LIN {X 0,Y 530.709,Z 614.143,A -85,B 0,C 180,E1 -4418.184,E2 -4418.184} C_VEL
LIN {X 0,Y 530.928,Z 606.171,A -85,B 0,C 180,E1 -4419.524,E2 -4419.524} C_VEL
LIN {X 0,Y 531.122,Z 597.851,A -85,B 0,C 180,E1 -4420.676,E2 -4420.676} C_VEL
LIN {X 0,Y 531.454,Z 587.351,A -85,B 0,C 180,E1 -4421.879,E2 -4421.879} C_VEL
LIN {X 0,Y 531.719,Z 576.624,A -85,B 0,C 180,E1 -4422.888,E2 -4422.888} C_VEL
LIN {X 0,Y 532.051,Z 564.106,A -85,B 0,C 180,E1 -4423.852,E2 -4423.852} C_VEL
LIN {X 0,Y 532.469,Z 551.67,A -85,B 0,C 180,E1 -4424.621,E2 -4424.621} C_VEL
LIN {X 0,Y 532.792,Z 537.759,A -85,B 0,C 180,E1 -4425.297,E2 -4425.297} C_VEL
LIN {X 0,Y 533.028,Z 523.286,A -85,B 0,C 180,E1 -4425.814,E2 -4425.814} C_VEL
LIN {X 0,Y 533.143,Z 514.195,A -85,B 0,C 180,E1 -4426.054,E2 -4426.054} C_VEL
LIN {X 0,Y 530.757,Z 502.42,A -85,B 0,C 180,E1 -4426.367,E2 -4426.367} C_VEL
LIN {X 0,Y 530.873,Z 494.542,A -85,B 0,C 180,E1 -4428.926,E2 -4428.926} C_VEL
LIN {X 0,Y 531.011,Z 485.976,A -85,B 0,C 180,E1 -4431.752,E2 -4431.752} C_VEL
LIN {X 0,Y 531.173,Z 477.41,A -85,B 0,C 180,E1 -4434.631,E2 -4434.631} C_VEL
LIN {X 0,Y 531.332,Z 470.067,A -85,B 0,C 180,E1 -4437.151,E2 -4437.151} C_VEL
LIN {X 0,Y 531.503,Z 463.949,A -85,B 0,C 180,E1 -4439.291,E2 -4439.291} C_VEL
LIN {X 0,Y 531.665,Z 455.312,A -85,B 0,C 180,E1 -4442.22,E2 -4442.22} C_VEL
LIN {X 0,Y 531.758,Z 447.204,A -85,B 0,C 180,E1 -4444.973,E2 -4444.973} C_VEL
LIN {X 0,Y 531.783,Z 438.711,A -85,B 0,C 180,E1 -4447.929,E2 -4447.929} C_VEL
LIN {X 0,Y 531.886,Z 429.937,A -85,B 0,C 180,E1 -4451.135,E2 -4451.135} C_VEL
LIN {X 0,Y 532.132,Z 421.148,A -85,B 0,C 180,E1 -4454.505,E2 -4454.505} C_VEL
LIN {X 0,Y 532.173,Z 415.877,A -85,B 0,C 180,E1 -4456.629,E2 -4456.629} C_VEL
LIN {X 0,Y 531.598,Z 411.207,A -85,B 0,C 180,E1 -4458.622,E2 -4458.622} C_VEL
LIN {X 0,Y 530.99,Z 407.971,A -85,B 0,C 180,E1 -4460.145,E2 -4460.145} C_VEL
LIN {X 0,Y 530.968,Z 407.972,A -85,B 0,C 180,E1 -4463.442,E2 -4463.442} C_VEL
LIN {X 0,Y 531.001,Z 407.967,A -85,B 0,C 180,E1 -4466.494,E2 -4466.494} C_VEL
LIN {X 0,Y 530.976,Z 407.969,A -85,B 0,C 180,E1 -4469.355,E2 -4469.355} C_VEL
LIN {X 0,Y 531.017,Z 407.964,A -85,B 0,C 180,E1 -4472.467,E2 -4472.467} C_VEL
LIN {X 0,Y 531.008,Z 407.963,A -85,B 0,C 180,E1 -4474.943,E2 -4474.943} C_VEL
LIN {X 0,Y 530.974,Z 407.967,A -85,B 0,C 180,E1 -4478.247,E2 -4478.247} C_VEL
LIN {X 0,Y 530.999,Z 407.967,A -85,B 0,C 180,E1 -4480.677,E2 -4480.677} C_VEL
LIN {X 0,Y 530.99,Z 407.968,A -85,B 0,C 180,E1 -4483.071,E2 -4483.071} C_VEL
LIN {X 0,Y 531.022,Z 407.959,A -85,B 0,C 180,E1 -4485.436,E2 -4485.436} C_VEL
LIN {X 0,Y 531.039,Z 407.96,A -85,B 0,C 180,E1 -4488.55,E2 -4488.55} C_VEL
LIN {X 0,Y 531.041,Z 407.957,A -85,B 0,C 180,E1 -4491.629,E2 -4491.629} C_VEL
LIN {X 0,Y 531.125,Z 407.95,A -85,B 0,C 180,E1 -4494.685,E2 -4494.685} C_VEL
LIN {X 0,Y 531.14,Z 407.944,A -85,B 0,C 180,E1 -4497.725,E2 -4497.725} C_VEL
LIN {X 0,Y 531.155,Z 407.946,A -85,B 0,C 180,E1 -4500.758,E2 -4500.758} C_VEL
LIN {X 0,Y 531.108,Z 407.951,A -85,B 0,C 180,E1 -4503.034,E2 -4503.034} C_VEL
LIN {X 0,Y 531.086,Z 407.959,A -85,B 0,C 180,E1 -4506.077,E2 -4506.077} C_VEL
LIN {X 0,Y 531.033,Z 407.962,A -85,B 0,C 180,E1 -4509.138,E2 -4509.138} C_VEL
LIN {X 0,Y 531.043,Z 407.962,A -85,B 0,C 180,E1 -4512.225,E2 -4512.225} C_VEL
LIN {X 0,Y 530.999,Z 407.968,A -85,B 0,C 180,E1 -4515.35,E2 -4515.35} C_VEL
LIN {X 0,Y 530.992,Z 407.964,A -85,B 0,C 180,E1 -4518.521,E2 -4518.521} C_VEL
LIN {X 0,Y 531.003,Z 407.969,A -85,B 0,C 180,E1 -4520.938,E2 -4520.938} C_VEL
LIN {X 0,Y 530.968,Z 407.973,A -85,B 0,C 180,E1 -4524.225,E2 -4524.225} C_VEL
LIN {X 0,Y 531.008,Z 407.964,A -85,B 0,C 180,E1 -4526.744,E2 -4526.744} C_VEL
LIN {X 0,Y 530.984,Z 407.967,A -85,B 0,C 180,E1 -4529.323,E2 -4529.323} C_VEL
LIN {X 0,Y 530.968,Z 407.97,A -85,B 0,C 180,E1 -4532.1,E2 -4532.1} C_VEL
LIN {X 0,Y 530.972,Z 407.971,A -85,B 0,C 180,E1 -4534.851,E2 -4534.851} C_VEL
LIN {X 0,Y 530.968,Z 407.974,A -85,B 0,C 180,E1 -4537.508,E2 -4537.508} C_VEL
LIN {X 0,Y 530.984,Z 407.971,A -85,B 0,C 180,E1 -4540.433,E2 -4540.433} C_VEL
LIN {X 0,Y 530.969,Z 407.973,A -85,B 0,C 180,E1 -4543.494,E2 -4543.494} C_VEL
LIN {X 0,Y 530.966,Z 407.973,A -85,B 0,C 180,E1 -4543.565,E2 -4543.565} C_VEL
LIN {X 0,Y 530.293,Z 408.054,A -85,B 0,C 180,E1 -4544.198,E2 -4544.198} C_VEL
LIN {X 0,Y 527.445,Z 408.413,A -85,B 0,C 180,E1 -4545.227,E2 -4545.227} C_VEL
LIN {X 0,Y 525.041,Z 408.716,A -85,B 0,C 180,E1 -4546.056,E2 -4546.056} C_VEL
LIN {X 0,Y 524.007,Z 408.843,A -85,B 0,C 180,E1 -4546.695,E2 -4546.695} C_VEL
LIN {X 0,Y 523.922,Z 408.852,A -85,B 0,C 180,E1 -4546.912,E2 -4546.912} C_VEL
LIN {X 0,Y 523.951,Z 408.848,A -85,B 0,C 180,E1 -4549.921,E2 -4549.921} C_VEL
LIN {X 0,Y 523.963,Z 408.854,A -85,B 0,C 180,E1 -4550.422,E2 -4550.422} C_VEL
LIN {X 0,Y 524.799,Z 414.518,A -85,B 0,C 180,E1 -4551.974,E2 -4551.974} C_VEL
LIN {X 0,Y 524.708,Z 423.272,A -85,B 0,C 180,E1 -4554.364,E2 -4554.364} C_VEL
LIN {X 0,Y 524.58,Z 434.74,A -85,B 0,C 180,E1 -4557.595,E2 -4557.595} C_VEL
LIN {X 0,Y 524.507,Z 445.196,A -85,B 0,C 180,E1 -4560.57,E2 -4560.57} C_VEL
LIN {X 0,Y 524.401,Z 454.996,A -85,B 0,C 180,E1 -4563.323,E2 -4563.323} C_VEL
LIN {X 0,Y 524.205,Z 465.688,A -85,B 0,C 180,E1 -4566.284,E2 -4566.284} C_VEL
LIN {X 0,Y 524.084,Z 476.206,A -85,B 0,C 180,E1 -4569.184,E2 -4569.184} C_VEL
LIN {X 0,Y 523.92,Z 487.271,A -85,B 0,C 180,E1 -4572.254,E2 -4572.254} C_VEL
LIN {X 0,Y 523.813,Z 491.641,A -85,B 0,C 180,E1 -4573.46,E2 -4573.46} C_VEL
LIN {X 0,Y 526.379,Z 504.566,A -85,B 0,C 180,E1 -4573.792,E2 -4573.792} C_VEL
LIN {X 0,Y 526.096,Z 519.046,A -85,B 0,C 180,E1 -4574.209,E2 -4574.209} C_VEL
LIN {X 0,Y 525.838,Z 532.206,A -85,B 0,C 180,E1 -4574.744,E2 -4574.744} C_VEL
LIN {X 0,Y 525.47,Z 545.972,A -85,B 0,C 180,E1 -4575.477,E2 -4575.477} C_VEL
LIN {X 0,Y 525.091,Z 557.559,A -85,B 0,C 180,E1 -4576.257,E2 -4576.257} C_VEL
LIN {X 0,Y 524.696,Z 569.44,A -85,B 0,C 180,E1 -4577.232,E2 -4577.232} C_VEL
LIN {X 0,Y 524.301,Z 580.988,A -85,B 0,C 180,E1 -4578.401,E2 -4578.401} C_VEL
LIN {X 0,Y 524.013,Z 590.481,A -85,B 0,C 180,E1 -4579.568,E2 -4579.568} C_VEL
LIN {X 0,Y 523.762,Z 599.542,A -85,B 0,C 180,E1 -4580.929,E2 -4580.929} C_VEL
LIN {X 0,Y 523.573,Z 606.843,A -85,B 0,C 180,E1 -4582.286,E2 -4582.286} C_VEL
LIN {X 0,Y 523.469,Z 613.433,A -85,B 0,C 180,E1 -4583.834,E2 -4583.834} C_VEL
LIN {X 0,Y 523.353,Z 618.327,A -85,B 0,C 180,E1 -4585.379,E2 -4585.379} C_VEL
LIN {X 0,Y 523.419,Z 620.227,A -85,B 0,C 180,E1 -4586.151,E2 -4586.151} C_VEL
LIN {X 0,Y 523.334,Z 622.94,A -85,B 0,C 180,E1 -4587.691,E2 -4587.691} C_VEL
LIN {X 0,Y 523.246,Z 624.299,A -85,B 0,C 180,E1 -4589.23,E2 -4589.23} C_VEL
LIN {X 0,Y 523.247,Z 624.346,A -85,B 0,C 180,E1 -4590.77,E2 -4590.77} C_VEL
LIN {X 0,Y 523.333,Z 623.049,A -85,B 0,C 180,E1 -4592.309,E2 -4592.309} C_VEL
LIN {X 0,Y 523.42,Z 620.43,A -85,B 0,C 180,E1 -4593.849,E2 -4593.849} C_VEL
LIN {X 0,Y 523.45,Z 616.35,A -85,B 0,C 180,E1 -4595.393,E2 -4595.393} C_VEL
LIN {X 0,Y 523.493,Z 612.29,A -85,B 0,C 180,E1 -4596.552,E2 -4596.552} C_VEL
LIN {X 0,Y 523.568,Z 607.269,A -85,B 0,C 180,E1 -4597.714,E2 -4597.714} C_VEL
LIN {X 0,Y 523.751,Z 600.085,A -85,B 0,C 180,E1 -4599.072,E2 -4599.072} C_VEL
LIN {X 0,Y 524.001,Z 591.128,A -85,B 0,C 180,E1 -4600.432,E2 -4600.432} C_VEL
LIN {X 0,Y 524.308,Z 581.8,A -85,B 0,C 180,E1 -4601.599,E2 -4601.599} C_VEL
LIN {X 0,Y 524.674,Z 570.39,A -85,B 0,C 180,E1 -4602.769,E2 -4602.769} C_VEL
LIN {X 0,Y 525.039,Z 558.753,A -85,B 0,C 180,E1 -4603.745,E2 -4603.745} C_VEL
LIN {X 0,Y 525.479,Z 545.827,A -85,B 0,C 180,E1 -4604.622,E2 -4604.622} C_VEL
LIN {X 0,Y 525.81,Z 532.013,A -85,B 0,C 180,E1 -4605.356,E2 -4605.356} C_VEL
LIN {X 0,Y 526.176,Z 517.48,A -85,B 0,C 180,E1 -4605.933,E2 -4605.933} C_VEL
LIN {X 0,Y 526.361,Z 504.166,A -85,B 0,C 180,E1 -4606.309,E2 -4606.309} C_VEL
LIN {X 0,Y 523.813,Z 491.588,A -85,B 0,C 180,E1 -4606.641,E2 -4606.641} C_VEL
LIN {X 0,Y 523.994,Z 480.988,A -85,B 0,C 180,E1 -4609.591,E2 -4609.591} C_VEL
LIN {X 0,Y 524.186,Z 470.27,A -85,B 0,C 180,E1 -4612.546,E2 -4612.546} C_VEL
LIN {X 0,Y 524.326,Z 458.655,A -85,B 0,C 180,E1 -4615.751,E2 -4615.751} C_VEL
LIN {X 0,Y 524.456,Z 449.135,A -85,B 0,C 180,E1 -4618.406,E2 -4618.406} C_VEL
LIN {X 0,Y 524.576,Z 438.248,A -85,B 0,C 180,E1 -4621.5,E2 -4621.5} C_VEL
LIN {X 0,Y 524.624,Z 428.598,A -85,B 0,C 180,E1 -4624.239,E2 -4624.239} C_VEL
LIN {X 0,Y 524.803,Z 418.429,A -85,B 0,C 180,E1 -4627.058,E2 -4627.058} C_VEL
LIN {X 0,Y 524.689,Z 413.124,A -85,B 0,C 180,E1 -4628.497,E2 -4628.497} C_VEL
LIN {X 0,Y 523.947,Z 408.849,A -85,B 0,C 180,E1 -4629.704,E2 -4629.704} C_VEL
LIN {X 0,Y 523.94,Z 408.849,A -85,B 0,C 180,E1 -4632.459,E2 -4632.459} C_VEL
LIN {X 0,Y 523.959,Z 408.846,A -85,B 0,C 180,E1 -4635.309,E2 -4635.309} C_VEL
LIN {X 0,Y 523.961,Z 408.847,A -85,B 0,C 180,E1 -4638.689,E2 -4638.689} C_VEL
LIN {X 0,Y 523.919,Z 408.851,A -85,B 0,C 180,E1 -4641.081,E2 -4641.081} C_VEL
LIN {X 0,Y 523.929,Z 408.848,A -85,B 0,C 180,E1 -4643.827,E2 -4643.827} C_VEL
LIN {X 0,Y 523.944,Z 408.846,A -85,B 0,C 180,E1 -4646.636,E2 -4646.636} C_VEL
LIN {X 0,Y 523.966,Z 408.84,A -85,B 0,C 180,E1 -4649.356,E2 -4649.356} C_VEL
LIN {X 0,Y 523.979,Z 408.842,A -85,B 0,C 180,E1 -4652.281,E2 -4652.281} C_VEL
LIN {X 0,Y 523.955,Z 408.844,A -85,B 0,C 180,E1 -4654.581,E2 -4654.581} C_VEL
LIN {X 0,Y 523.92,Z 408.849,A -85,B 0,C 180,E1 -4657.107,E2 -4657.107} C_VEL
LIN {X 0,Y 523.982,Z 408.845,A -85,B 0,C 180,E1 -4659.866,E2 -4659.866} C_VEL
LIN {X 0,Y 523.963,Z 408.851,A -85,B 0,C 180,E1 -4661.417,E2 -4661.417} C_VEL
LIN {X 0,Y 526.697,Z 417.552,A -85,B 0,C 180,E1 -4661.826,E2 -4661.826} C_VEL
LIN {X 0,Y 526.634,Z 428.886,A -85,B 0,C 180,E1 -4662.326,E2 -4662.326} C_VEL
LIN {X 0,Y 526.283,Z 440.14,A -85,B 0,C 180,E1 -4662.915,E2 -4662.915} C_VEL
LIN {X 0,Y 525.888,Z 451.09,A -85,B 0,C 180,E1 -4663.601,E2 -4663.601} C_VEL
LIN {X 0,Y 525.483,Z 461.333,A -85,B 0,C 180,E1 -4664.356,E2 -4664.356} C_VEL
LIN {X 0,Y 525.097,Z 470.829,A -85,B 0,C 180,E1 -4665.17,E2 -4665.17} C_VEL
LIN {X 0,Y 524.748,Z 479.724,A -85,B 0,C 180,E1 -4666.05,E2 -4666.05} C_VEL
LIN {X 0,Y 524.46,Z 488.326,A -85,B 0,C 180,E1 -4667.029,E2 -4667.029} C_VEL
LIN {X 0,Y 524.085,Z 497.442,A -85,B 0,C 180,E1 -4668.219,E2 -4668.219} C_VEL
LIN {X 0,Y 523.917,Z 506.187,A -85,B 0,C 180,E1 -4669.566,E2 -4669.566} C_VEL
LIN {X 0,Y 523.66,Z 514.361,A -85,B 0,C 180,E1 -4671.121,E2 -4671.121} C_VEL
LIN {X 0,Y 523.546,Z 519.47,A -85,B 0,C 180,E1 -4672.285,E2 -4672.285} C_VEL
LIN {X 0,Y 523.467,Z 523.823,A -85,B 0,C 180,E1 -4673.472,E2 -4673.472} C_VEL
LIN {X 0,Y 523.441,Z 527.259,A -85,B 0,C 180,E1 -4674.607,E2 -4674.607} C_VEL
LIN {X 0,Y 523.402,Z 530.761,A -85,B 0,C 180,E1 -4676.15,E2 -4676.15} C_VEL
LIN {X 0,Y 523.359,Z 532.149,A -85,B 0,C 180,E1 -4676.921,E2 -4676.921} C_VEL
LIN {X 0,Y 523.27,Z 533.858,A -85,B 0,C 180,E1 -4678.461,E2 -4678.461} C_VEL
LIN {X 0,Y 523.244,Z 534.43,A -85,B 0,C 180,E1 -4680,E2 -4680} C_VEL
LIN {X 0,Y 523.248,Z 534.369,A -85,B 0,C 180,E1 -4680.77,E2 -4680.77} C_VEL
LIN {X 0,Y 523.332,Z 533.247,A -85,B 0,C 180,E1 -4682.309,E2 -4682.309} C_VEL
LIN {X 0,Y 523.403,Z 530.941,A -85,B 0,C 180,E1 -4683.85,E2 -4683.85} C_VEL
LIN {X 0,Y 523.322,Z 529.424,A -85,B 0,C 180,E1 -4684.622,E2 -4684.622} C_VEL
LIN {X 0,Y 523.447,Z 525.299,A -85,B 0,C 180,E1 -4686.166,E2 -4686.166} C_VEL
LIN {X 0,Y 523.533,Z 519.815,A -85,B 0,C 180,E1 -4687.715,E2 -4687.715} C_VEL
LIN {X 0,Y 523.643,Z 514.778,A -85,B 0,C 180,E1 -4688.879,E2 -4688.879} C_VEL
LIN {X 0,Y 523.773,Z 508.825,A -85,B 0,C 180,E1 -4690.046,E2 -4690.046} C_VEL
LIN {X 0,Y 524.03,Z 501.839,A -85,B 0,C 180,E1 -4691.213,E2 -4691.213} C_VEL
LIN {X 0,Y 524.203,Z 495.095,A -85,B 0,C 180,E1 -4692.194,E2 -4692.194} C_VEL
LIN {X 0,Y 524.48,Z 487.449,A -85,B 0,C 180,E1 -4693.167,E2 -4693.167} C_VEL
LIN {X 0,Y 524.814,Z 478.744,A -85,B 0,C 180,E1 -4694.146,E2 -4694.146} C_VEL
LIN {X 0,Y 525.139,Z 469.8,A -85,B 0,C 180,E1 -4695.019,E2 -4695.019} C_VEL
LIN {X 0,Y 525.609,Z 459.629,A -85,B 0,C 180,E1 -4695.869,E2 -4695.869} C_VEL
LIN {X 0,Y 525.986,Z 448.044,A -85,B 0,C 180,E1 -4696.695,E2 -4696.695} C_VEL
LIN {X 0,Y 526.476,Z 434.632,A -85,B 0,C 180,E1 -4697.479,E2 -4697.479} C_VEL
LIN {X 0,Y 526.827,Z 420.353,A -85,B 0,C 180,E1 -4698.132,E2 -4698.132} C_VEL
LIN {X 0,Y 526.605,Z 417.439,A -85,B 0,C 180,E1 -4698.258,E2 -4698.258} C_VEL
LIN {X 0,Y 523.963,Z 408.843,A -85,B 0,C 180,E1 -4698.655,E2 -4698.655} C_VEL
LIN {X 0,Y 523.948,Z 408.843,A -85,B 0,C 180,E1 -4701.233,E2 -4701.233} C_VEL
LIN {X 0,Y 523.928,Z 408.847,A -85,B 0,C 180,E1 -4704.572,E2 -4704.572} C_VEL
LIN {X 0,Y 523.956,Z 408.842,A -85,B 0,C 180,E1 -4707.133,E2 -4707.133} C_VEL
LIN {X 0,Y 523.945,Z 408.849,A -85,B 0,C 180,E1 -4709.756,E2 -4709.756} C_VEL
LIN {X 0,Y 523.942,Z 408.843,A -85,B 0,C 180,E1 -4712.449,E2 -4712.449} C_VEL
LIN {X 0,Y 523.922,Z 408.847,A -85,B 0,C 180,E1 -4715.227,E2 -4715.227} C_VEL
LIN {X 0,Y 523.917,Z 408.849,A -85,B 0,C 180,E1 -4718.102,E2 -4718.102} C_VEL
LIN {X 0,Y 523.943,Z 408.845,A -85,B 0,C 180,E1 -4721.092,E2 -4721.092} C_VEL
LIN {X 0,Y 523.952,Z 408.846,A -85,B 0,C 180,E1 -4724.227,E2 -4724.227} C_VEL
LIN {X 0,Y 523.997,Z 408.934,A -85,B 0,C 180,E1 -4724.797,E2 -4724.797} C_VEL
LIN {X 0,Y 523.747,Z 419.256,A -85,B 0,C 180,E1 -4727.861,E2 -4727.861} C_VEL
LIN {X 0,Y 524.048,Z 430.498,A -85,B 0,C 180,E1 -4731.063,E2 -4731.063} C_VEL
LIN {X 0,Y 524.288,Z 440.494,A -85,B 0,C 180,E1 -4733.856,E2 -4733.856} C_VEL
LIN {X 0,Y 524.4,Z 448.893,A -85,B 0,C 180,E1 -4736.194,E2 -4736.194} C_VEL
LIN {X 0,Y 524.489,Z 459.131,A -85,B 0,C 180,E1 -4739.046,E2 -4739.046} C_VEL
LIN {X 0,Y 524.528,Z 466.39,A -85,B 0,C 180,E1 -4741.161,E2 -4741.161} C_VEL
LIN {X 0,Y 524.219,Z 476.186,A -85,B 0,C 180,E1 -4744.595,E2 -4744.595} C_VEL
LIN {X 0,Y 523.984,Z 485.381,A -85,B 0,C 180,E1 -4747.74,E2 -4747.74} C_VEL
LIN {X 0,Y 523.869,Z 493.319,A -85,B 0,C 180,E1 -4750.404,E2 -4750.404} C_VEL
LIN {X 0,Y 523.742,Z 502.599,A -85,B 0,C 180,E1 -4753.432,E2 -4753.432} C_VEL
LIN {X 0,Y 526.393,Z 515.813,A -85,B 0,C 180,E1 -4753.774,E2 -4753.774} C_VEL
LIN {X 0,Y 526.109,Z 529.055,A -85,B 0,C 180,E1 -4754.162,E2 -4754.162} C_VEL
LIN {X 0,Y 525.793,Z 543.152,A -85,B 0,C 180,E1 -4754.743,E2 -4754.743} C_VEL
LIN {X 0,Y 525.438,Z 556.679,A -85,B 0,C 180,E1 -4755.476,E2 -4755.476} C_VEL
LIN {X 0,Y 525.001,Z 569.459,A -85,B 0,C 180,E1 -4756.353,E2 -4756.353} C_VEL
LIN {X 0,Y 524.624,Z 580.966,A -85,B 0,C 180,E1 -4757.328,E2 -4757.328} C_VEL
LIN {X 0,Y 524.335,Z 591.384,A -85,B 0,C 180,E1 -4758.401,E2 -4758.401} C_VEL
LIN {X 0,Y 523.997,Z 600.801,A -85,B 0,C 180,E1 -4759.568,E2 -4759.568} C_VEL
LIN {X 0,Y 523.761,Z 609.812,A -85,B 0,C 180,E1 -4760.929,E2 -4760.929} C_VEL
LIN {X 0,Y 523.569,Z 617.068,A -85,B 0,C 180,E1 -4762.286,E2 -4762.286} C_VEL
LIN {X 0,Y 523.468,Z 623.582,A -85,B 0,C 180,E1 -4763.834,E2 -4763.834} C_VEL
LIN {X 0,Y 523.376,Z 627.394,A -85,B 0,C 180,E1 -4764.993,E2 -4764.993} C_VEL
LIN {X 0,Y 523.419,Z 630.314,A -85,B 0,C 180,E1 -4766.151,E2 -4766.151} C_VEL
LIN {X 0,Y 523.333,Z 632.997,A -85,B 0,C 180,E1 -4767.691,E2 -4767.691} C_VEL
LIN {X 0,Y 523.247,Z 634.332,A -85,B 0,C 180,E1 -4769.23,E2 -4769.23} C_VEL
LIN {X 0,Y 523.247,Z 634.331,A -85,B 0,C 180,E1 -4770.77,E2 -4770.77} C_VEL
LIN {X 0,Y 523.333,Z 632.997,A -85,B 0,C 180,E1 -4772.309,E2 -4772.309} C_VEL
LIN {X 0,Y 523.419,Z 630.318,A -85,B 0,C 180,E1 -4773.849,E2 -4773.849} C_VEL
LIN {X 0,Y 523.449,Z 626.217,A -85,B 0,C 180,E1 -4775.393,E2 -4775.393} C_VEL
LIN {X 0,Y 523.495,Z 620.547,A -85,B 0,C 180,E1 -4776.94,E2 -4776.94} C_VEL
LIN {X 0,Y 523.664,Z 614.145,A -85,B 0,C 180,E1 -4778.295,E2 -4778.295} C_VEL
LIN {X 0,Y 523.863,Z 606.17,A -85,B 0,C 180,E1 -4779.654,E2 -4779.654} C_VEL
LIN {X 0,Y 524.115,Z 597.851,A -85,B 0,C 180,E1 -4780.82,E2 -4780.82} C_VEL
LIN {X 0,Y 524.449,Z 587.082,A -85,B 0,C 180,E1 -4782.068,E2 -4782.068} C_VEL
LIN {X 0,Y 524.805,Z 575.469,A -85,B 0,C 180,E1 -4783.159,E2 -4783.159} C_VEL
LIN {X 0,Y 525.179,Z 562.703,A -85,B 0,C 180,E1 -4784.136,E2 -4784.136} C_VEL
LIN {X 0,Y 525.639,Z 549.923,A -85,B 0,C 180,E1 -4784.915,E2 -4784.915} C_VEL
LIN {X 0,Y 525.937,Z 537.761,A -85,B 0,C 180,E1 -4785.501,E2 -4785.501} C_VEL
LIN {X 0,Y 526.206,Z 523.168,A -85,B 0,C 180,E1 -4786.028,E2 -4786.028} C_VEL
LIN {X 0,Y 526.212,Z 514.561,A -85,B 0,C 180,E1 -4786.263,E2 -4786.263} C_VEL
LIN {X 0,Y 523.732,Z 502.42,A -85,B 0,C 180,E1 -4786.593,E2 -4786.593} C_VEL
LIN {X 0,Y 523.869,Z 493.319,A -85,B 0,C 180,E1 -4789.596,E2 -4789.596} C_VEL
LIN {X 0,Y 523.984,Z 485.381,A -85,B 0,C 180,E1 -4792.26,E2 -4792.26} C_VEL
LIN {X 0,Y 524.219,Z 476.186,A -85,B 0,C 180,E1 -4795.405,E2 -4795.405} C_VEL
LIN {X 0,Y 524.528,Z 466.39,A -85,B 0,C 180,E1 -4798.839,E2 -4798.839} C_VEL
LIN {X 0,Y 524.587,Z 457.054,A -85,B 0,C 180,E1 -4801.951,E2 -4801.951} C_VEL
LIN {X 0,Y 524.695,Z 449.048,A -85,B 0,C 180,E1 -4804.699,E2 -4804.699} C_VEL
LIN {X 0,Y 524.763,Z 441.282,A -85,B 0,C 180,E1 -4807.432,E2 -4807.432} C_VEL
LIN {X 0,Y 524.879,Z 433.589,A -85,B 0,C 180,E1 -4810.251,E2 -4810.251} C_VEL
LIN {X 0,Y 524.991,Z 426.262,A -85,B 0,C 180,E1 -4813.058,E2 -4813.058} C_VEL
LIN {X 0,Y 525.253,Z 419.101,A -85,B 0,C 180,E1 -4815.911,E2 -4815.911} C_VEL
LIN {X 0,Y 525.086,Z 415.535,A -85,B 0,C 180,E1 -4817.404,E2 -4817.404} C_VEL
LIN {X 0,Y 524.13,Z 409.809,A -85,B 0,C 180,E1 -4819.937,E2 -4819.937} C_VEL
LIN {X 0,Y 523.95,Z 408.848,A -85,B 0,C 180,E1 -4820.421,E2 -4820.421} C_VEL
LIN {X 0,Y 523.922,Z 408.85,A -85,B 0,C 180,E1 -4823.596,E2 -4823.596} C_VEL
LIN {X 0,Y 523.943,Z 408.847,A -85,B 0,C 180,E1 -4826.636,E2 -4826.636} C_VEL
LIN {X 0,Y 523.957,Z 408.844,A -85,B 0,C 180,E1 -4829.356,E2 -4829.356} C_VEL
LIN {X 0,Y 523.981,Z 408.84,A -85,B 0,C 180,E1 -4832.281,E2 -4832.281} C_VEL
LIN {X 0,Y 523.956,Z 408.844,A -85,B 0,C 180,E1 -4834.581,E2 -4834.581} C_VEL
LIN {X 0,Y 523.92,Z 408.849,A -85,B 0,C 180,E1 -4837.107,E2 -4837.107} C_VEL
LIN {X 0,Y 523.981,Z 408.835,A -85,B 0,C 180,E1 -4839.866,E2 -4839.866} C_VEL
LIN {X 0,Y 523.97,Z 408.841,A -85,B 0,C 180,E1 -4842.837,E2 -4842.837} C_VEL
LIN {X 0,Y 523.979,Z 408.838,A -85,B 0,C 180,E1 -4845.236,E2 -4845.236} C_VEL
LIN {X 0,Y 524.015,Z 408.836,A -85,B 0,C 180,E1 -4848.394,E2 -4848.394} C_VEL
LIN {X 0,Y 523.993,Z 408.834,A -85,B 0,C 180,E1 -4851.516,E2 -4851.516} C_VEL
LIN {X 0,Y 524.086,Z 408.826,A -85,B 0,C 180,E1 -4854.614,E2 -4854.614} C_VEL
LIN {X 0,Y 524.112,Z 408.819,A -85,B 0,C 180,E1 -4857.695,E2 -4857.695} C_VEL
LIN {X 0,Y 524.126,Z 408.821,A -85,B 0,C 180,E1 -4860.768,E2 -4860.768} C_VEL
LIN {X 0,Y 524.074,Z 408.827,A -85,B 0,C 180,E1 -4863.075,E2 -4863.075} C_VEL
LIN {X 0,Y 524.048,Z 408.834,A -85,B 0,C 180,E1 -4866.159,E2 -4866.159} C_VEL
LIN {X 0,Y 524.001,Z 408.838,A -85,B 0,C 180,E1 -4869.262,E2 -4869.262} C_VEL
LIN {X 0,Y 524.005,Z 408.839,A -85,B 0,C 180,E1 -4871.74,E2 -4871.74} C_VEL
LIN {X 0,Y 523.996,Z 408.841,A -85,B 0,C 180,E1 -4875.052,E2 -4875.052} C_VEL
LIN {X 0,Y 523.966,Z 408.844,A -85,B 0,C 180,E1 -4877.969,E2 -4877.969} C_VEL
LIN {X 0,Y 523.975,Z 408.841,A -85,B 0,C 180,E1 -4880.41,E2 -4880.41} C_VEL
LIN {X 0,Y 523.913,Z 408.848,A -85,B 0,C 180,E1 -4882.894,E2 -4882.894} C_VEL
LIN {X 0,Y 523.987,Z 408.838,A -85,B 0,C 180,E1 -4886.02,E2 -4886.02} C_VEL
LIN {X 0,Y 523.942,Z 408.846,A -85,B 0,C 180,E1 -4888.875,E2 -4888.875} C_VEL
LIN {X 0,Y 523.924,Z 408.852,A -85,B 0,C 180,E1 -4891.544,E2 -4891.544} C_VEL
LIN {X 0,Y 523.935,Z 408.847,A -85,B 0,C 180,E1 -4894.29,E2 -4894.29} C_VEL
LIN {X 0,Y 523.909,Z 408.85,A -85,B 0,C 180,E1 -4897.132,E2 -4897.132} C_VEL
LIN {X 0,Y 523.939,Z 408.846,A -85,B 0,C 180,E1 -4900.13,E2 -4900.13} C_VEL
LIN {X 0,Y 523.942,Z 408.847,A -85,B 0,C 180,E1 -4902.459,E2 -4902.459} C_VEL
LIN {X 0,Y 523.959,Z 408.847,A -85,B 0,C 180,E1 -4905.309,E2 -4905.309} C_VEL
LIN {X 0,Y 523.922,Z 408.852,A -85,B 0,C 180,E1 -4906.912,E2 -4906.912} C_VEL
LIN {X 0,Y 523.241,Z 408.936,A -85,B 0,C 180,E1 -4907.34,E2 -4907.34} C_VEL
LIN {X 0,Y 520.398,Z 409.293,A -85,B 0,C 180,E1 -4908.009,E2 -4908.009} C_VEL
LIN {X 0,Y 517.552,Z 409.647,A -85,B 0,C 180,E1 -4908.684,E2 -4908.684} C_VEL
LIN {X 0,Y 516.884,Z 409.729,A -85,B 0,C 180,E1 -4909.12,E2 -4909.12} C_VEL
LIN {X 0,Y 516.955,Z 409.896,A -85,B 0,C 180,E1 -4910.285,E2 -4910.285} C_VEL
LIN {X 0,Y 517.853,Z 415.763,A -85,B 0,C 180,E1 -4911.919,E2 -4911.919} C_VEL
LIN {X 0,Y 517.725,Z 425.224,A -85,B 0,C 180,E1 -4914.537,E2 -4914.537} C_VEL
LIN {X 0,Y 517.577,Z 437.464,A -85,B 0,C 180,E1 -4918.024,E2 -4918.024} C_VEL
LIN {X 0,Y 517.455,Z 446.879,A -85,B 0,C 180,E1 -4920.729,E2 -4920.729} C_VEL
LIN {X 0,Y 517.373,Z 454.607,A -85,B 0,C 180,E1 -4922.931,E2 -4922.931} C_VEL
LIN {X 0,Y 517.176,Z 465.383,A -85,B 0,C 180,E1 -4925.941,E2 -4925.941} C_VEL
LIN {X 0,Y 517.082,Z 474.488,A -85,B 0,C 180,E1 -4928.471,E2 -4928.471} C_VEL
LIN {X 0,Y 516.923,Z 484.937,A -85,B 0,C 180,E1 -4931.367,E2 -4931.367} C_VEL
LIN {X 0,Y 516.779,Z 491.628,A -85,B 0,C 180,E1 -4933.228,E2 -4933.228} C_VEL
LIN {X 0,Y 519.536,Z 505.622,A -85,B 0,C 180,E1 -4933.598,E2 -4933.598} C_VEL
LIN {X 0,Y 519.262,Z 519.612,A -85,B 0,C 180,E1 -4934.015,E2 -4934.015} C_VEL
LIN {X 0,Y 518.954,Z 533.309,A -85,B 0,C 180,E1 -4934.587,E2 -4934.587} C_VEL
LIN {X 0,Y 518.575,Z 546.012,A -85,B 0,C 180,E1 -4935.279,E2 -4935.279} C_VEL
LIN {X 0,Y 518.169,Z 557.633,A -85,B 0,C 180,E1 -4936.069,E2 -4936.069} C_VEL
LIN {X 0,Y 517.732,Z 569.449,A -85,B 0,C 180,E1 -4937.057,E2 -4937.057} C_VEL
LIN {X 0,Y 517.295,Z 580.345,A -85,B 0,C 180,E1 -4938.167,E2 -4938.167} C_VEL
LIN {X 0,Y 517.013,Z 590.492,A -85,B 0,C 180,E1 -4939.426,E2 -4939.426} C_VEL
LIN {X 0,Y 516.731,Z 599.547,A -85,B 0,C 180,E1 -4940.804,E2 -4940.804} C_VEL
LIN {X 0,Y 516.506,Z 606.846,A -85,B 0,C 180,E1 -4942.18,E2 -4942.18} C_VEL
LIN {X 0,Y 516.385,Z 613.437,A -85,B 0,C 180,E1 -4943.749,E2 -4943.749} C_VEL
LIN {X 0,Y 516.306,Z 617.266,A -85,B 0,C 180,E1 -4944.924,E2 -4944.924} C_VEL
LIN {X 0,Y 516.325,Z 620.228,A -85,B 0,C 180,E1 -4946.098,E2 -4946.098} C_VEL
LIN {X 0,Y 516.26,Z 622.939,A -85,B 0,C 180,E1 -4947.659,E2 -4947.659} C_VEL
LIN {X 0,Y 516.156,Z 624.298,A -85,B 0,C 180,E1 -4949.22,E2 -4949.22} C_VEL
LIN {X 0,Y 516.157,Z 624.345,A -85,B 0,C 180,E1 -4950.78,E2 -4950.78} C_VEL
LIN {X 0,Y 516.259,Z 623.046,A -85,B 0,C 180,E1 -4952.341,E2 -4952.341} C_VEL
LIN {X 0,Y 516.325,Z 620.429,A -85,B 0,C 180,E1 -4953.902,E2 -4953.902} C_VEL
LIN {X 0,Y 516.384,Z 616.347,A -85,B 0,C 180,E1 -4955.467,E2 -4955.467} C_VEL
LIN {X 0,Y 516.398,Z 612.708,A -85,B 0,C 180,E1 -4956.533,E2 -4956.533} C_VEL
LIN {X 0,Y 516.499,Z 607.266,A -85,B 0,C 180,E1 -4957.821,E2 -4957.821} C_VEL
LIN {X 0,Y 516.701,Z 600.083,A -85,B 0,C 180,E1 -4959.196,E2 -4959.196} C_VEL
LIN {X 0,Y 516.996,Z 591.153,A -85,B 0,C 180,E1 -4960.575,E2 -4960.575} C_VEL
LIN {X 0,Y 517.326,Z 580.986,A -85,B 0,C 180,E1 -4961.849,E2 -4961.849} C_VEL
LIN {X 0,Y 517.724,Z 570.392,A -85,B 0,C 180,E1 -4962.943,E2 -4962.943} C_VEL
LIN {X 0,Y 518.094,Z 558.767,A -85,B 0,C 180,E1 -4963.933,E2 -4963.933} C_VEL
LIN {X 0,Y 518.537,Z 547.395,A -85,B 0,C 180,E1 -4964.722,E2 -4964.722} C_VEL
LIN {X 0,Y 518.921,Z 534.135,A -85,B 0,C 180,E1 -4965.464,E2 -4965.464} C_VEL
LIN {X 0,Y 519.249,Z 521.235,A -85,B 0,C 180,E1 -4966.018,E2 -4966.018} C_VEL
LIN {X 0,Y 519.559,Z 506.851,A -85,B 0,C 180,E1 -4966.462,E2 -4966.462} C_VEL
LIN {X 0,Y 518.68,Z 500.619,A -85,B 0,C 180,E1 -4966.635,E2 -4966.635} C_VEL
LIN {X 0,Y 516.806,Z 491.575,A -85,B 0,C 180,E1 -4966.873,E2 -4966.873} C_VEL
LIN {X 0,Y 516.987,Z 480.828,A -85,B 0,C 180,E1 -4969.868,E2 -4969.868} C_VEL
LIN {X 0,Y 517.143,Z 470.286,A -85,B 0,C 180,E1 -4972.787,E2 -4972.787} C_VEL
LIN {X 0,Y 517.281,Z 459.55,A -85,B 0,C 180,E1 -4975.77,E2 -4975.77} C_VEL
LIN {X 0,Y 517.439,Z 450.29,A -85,B 0,C 180,E1 -4978.384,E2 -4978.384} C_VEL
LIN {X 0,Y 517.55,Z 440.547,A -85,B 0,C 180,E1 -4981.185,E2 -4981.185} C_VEL
LIN {X 0,Y 517.632,Z 429.382,A -85,B 0,C 180,E1 -4984.382,E2 -4984.382} C_VEL
LIN {X 0,Y 517.85,Z 419.401,A -85,B 0,C 180,E1 -4987.175,E2 -4987.175} C_VEL
LIN {X 0,Y 517.653,Z 414.051,A -85,B 0,C 180,E1 -4988.648,E2 -4988.648} C_VEL
LIN {X 0,Y 516.895,Z 409.728,A -85,B 0,C 180,E1 -4989.908,E2 -4989.908} C_VEL
LIN {X 0,Y 516.887,Z 409.727,A -85,B 0,C 180,E1 -4992.831,E2 -4992.831} C_VEL
LIN {X 0,Y 516.925,Z 409.723,A -85,B 0,C 180,E1 -4995.01,E2 -4995.01} C_VEL
LIN {X 0,Y 516.918,Z 409.725,A -85,B 0,C 180,E1 -4998.398,E2 -4998.398} C_VEL
LIN {X 0,Y 516.882,Z 409.727,A -85,B 0,C 180,E1 -5001.284,E2 -5001.284} C_VEL
LIN {X 0,Y 516.891,Z 409.727,A -85,B 0,C 180,E1 -5004.221,E2 -5004.221} C_VEL
LIN {X 0,Y 516.897,Z 409.724,A -85,B 0,C 180,E1 -5007.053,E2 -5007.053} C_VEL
LIN {X 0,Y 516.903,Z 409.719,A -85,B 0,C 180,E1 -5009.797,E2 -5009.797} C_VEL
LIN {X 0,Y 516.928,Z 409.722,A -85,B 0,C 180,E1 -5012.467,E2 -5012.467} C_VEL
LIN {X 0,Y 516.913,Z 409.724,A -85,B 0,C 180,E1 -5015.072,E2 -5015.072} C_VEL
LIN {X 0,Y 516.873,Z 409.729,A -85,B 0,C 180,E1 -5017.622,E2 -5017.622} C_VEL
LIN {X 0,Y 516.935,Z 409.722,A -85,B 0,C 180,E1 -5020.13,E2 -5020.13} C_VEL
LIN {X 0,Y 516.944,Z 409.786,A -85,B 0,C 180,E1 -5021.195,E2 -5021.195} C_VEL
LIN {X 0,Y 520.053,Z 419.942,A -85,B 0,C 180,E1 -5021.687,E2 -5021.687} C_VEL
LIN {X 0,Y 519.749,Z 432.987,A -85,B 0,C 180,E1 -5022.287,E2 -5022.287} C_VEL
LIN {X 0,Y 519.248,Z 446.951,A -85,B 0,C 180,E1 -5023.082,E2 -5023.082} C_VEL
LIN {X 0,Y 518.741,Z 460.065,A -85,B 0,C 180,E1 -5024.015,E2 -5024.015} C_VEL
LIN {X 0,Y 518.268,Z 470.326,A -85,B 0,C 180,E1 -5024.886,E2 -5024.886} C_VEL
LIN {X 0,Y 517.865,Z 480.169,A -85,B 0,C 180,E1 -5025.861,E2 -5025.861} C_VEL
LIN {X 0,Y 517.553,Z 488.779,A -85,B 0,C 180,E1 -5026.853,E2 -5026.853} C_VEL
LIN {X 0,Y 517.201,Z 496.275,A -85,B 0,C 180,E1 -5027.841,E2 -5027.841} C_VEL
LIN {X 0,Y 517.026,Z 502.798,A -85,B 0,C 180,E1 -5028.831,E2 -5028.831} C_VEL
LIN {X 0,Y 516.714,Z 509.564,A -85,B 0,C 180,E1 -5030.013,E2 -5030.013} C_VEL
LIN {X 0,Y 516.599,Z 514.424,A -85,B 0,C 180,E1 -5030.999,E2 -5030.999} C_VEL
LIN {X 0,Y 516.473,Z 519.465,A -85,B 0,C 180,E1 -5032.179,E2 -5032.179} C_VEL
LIN {X 0,Y 516.371,Z 524.168,A -85,B 0,C 180,E1 -5033.493,E2 -5033.493} C_VEL
LIN {X 0,Y 516.373,Z 527.254,A -85,B 0,C 180,E1 -5034.533,E2 -5034.533} C_VEL
LIN {X 0,Y 516.308,Z 530.758,A -85,B 0,C 180,E1 -5036.097,E2 -5036.097} C_VEL
LIN {X 0,Y 516.272,Z 532.152,A -85,B 0,C 180,E1 -5036.879,E2 -5036.879} C_VEL
LIN {X 0,Y 516.188,Z 533.854,A -85,B 0,C 180,E1 -5038.44,E2 -5038.44} C_VEL
LIN {X 0,Y 516.152,Z 534.424,A -85,B 0,C 180,E1 -5040,E2 -5040} C_VEL
LIN {X 0,Y 516.158,Z 534.37,A -85,B 0,C 180,E1 -5040.78,E2 -5040.78} C_VEL
LIN {X 0,Y 516.258,Z 533.24,A -85,B 0,C 180,E1 -5042.341,E2 -5042.341} C_VEL
LIN {X 0,Y 516.308,Z 530.934,A -85,B 0,C 180,E1 -5043.903,E2 -5043.903} C_VEL
LIN {X 0,Y 516.238,Z 529.421,A -85,B 0,C 180,E1 -5044.685,E2 -5044.685} C_VEL
LIN {X 0,Y 516.372,Z 525.291,A -85,B 0,C 180,E1 -5046.251,E2 -5046.251} C_VEL
LIN {X 0,Y 516.461,Z 519.807,A -85,B 0,C 180,E1 -5047.821,E2 -5047.821} C_VEL
LIN {X 0,Y 516.579,Z 514.853,A -85,B 0,C 180,E1 -5049.001,E2 -5049.001} C_VEL
LIN {X 0,Y 516.755,Z 509.049,A -85,B 0,C 180,E1 -5050.184,E2 -5050.184} C_VEL
LIN {X 0,Y 517.035,Z 502.21,A -85,B 0,C 180,E1 -5051.367,E2 -5051.367} C_VEL
LIN {X 0,Y 517.304,Z 494.187,A -85,B 0,C 180,E1 -5052.555,E2 -5052.555} C_VEL
LIN {X 0,Y 517.723,Z 484.75,A -85,B 0,C 180,E1 -5053.742,E2 -5053.742} C_VEL
LIN {X 0,Y 518.157,Z 473.391,A -85,B 0,C 180,E1 -5054.934,E2 -5054.934} C_VEL
LIN {X 0,Y 518.669,Z 462.264,A -85,B 0,C 180,E1 -5055.905,E2 -5055.905} C_VEL
LIN {X 0,Y 519.123,Z 449.772,A -85,B 0,C 180,E1 -5056.821,E2 -5056.821} C_VEL
LIN {X 0,Y 519.599,Z 436.495,A -85,B 0,C 180,E1 -5057.616,E2 -5057.616} C_VEL
LIN {X 0,Y 519.977,Z 422.263,A -85,B 0,C 180,E1 -5058.288,E2 -5058.288} C_VEL
LIN {X 0,Y 519.934,Z 419.564,A -85,B 0,C 180,E1 -5058.401,E2 -5058.401} C_VEL
LIN {X 0,Y 516.916,Z 409.72,A -85,B 0,C 180,E1 -5058.867,E2 -5058.867} C_VEL
LIN {X 0,Y 516.888,Z 409.725,A -85,B 0,C 180,E1 -5061.538,E2 -5061.538} C_VEL
LIN {X 0,Y 516.884,Z 409.727,A -85,B 0,C 180,E1 -5064.357,E2 -5064.357} C_VEL
LIN {X 0,Y 516.929,Z 409.718,A -85,B 0,C 180,E1 -5066.658,E2 -5066.658} C_VEL
LIN {X 0,Y 516.913,Z 409.724,A -85,B 0,C 180,E1 -5069.524,E2 -5069.524} C_VEL
LIN {X 0,Y 516.903,Z 409.72,A -85,B 0,C 180,E1 -5072.544,E2 -5072.544} C_VEL
LIN {X 0,Y 516.868,Z 409.727,A -85,B 0,C 180,E1 -5075.33,E2 -5075.33} C_VEL
LIN {X 0,Y 516.882,Z 409.727,A -85,B 0,C 180,E1 -5077.943,E2 -5077.943} C_VEL
LIN {X 0,Y 516.886,Z 409.722,A -85,B 0,C 180,E1 -5080.741,E2 -5080.741} C_VEL
LIN {X 0,Y 516.907,Z 409.722,A -85,B 0,C 180,E1 -5082.829,E2 -5082.829} C_VEL
LIN {X 0,Y 516.966,Z 409.844,A -85,B 0,C 180,E1 -5084.711,E2 -5084.711} C_VEL
LIN {X 0,Y 516.708,Z 418.142,A -85,B 0,C 180,E1 -5087.263,E2 -5087.263} C_VEL
LIN {X 0,Y 516.956,Z 430.227,A -85,B 0,C 180,E1 -5090.797,E2 -5090.797} C_VEL
LIN {X 0,Y 517.22,Z 440.677,A -85,B 0,C 180,E1 -5093.776,E2 -5093.776} C_VEL
LIN {X 0,Y 517.333,Z 450.747,A -85,B 0,C 180,E1 -5096.62,E2 -5096.62} C_VEL
LIN {X 0,Y 517.385,Z 460.518,A -85,B 0,C 180,E1 -5099.377,E2 -5099.377} C_VEL
LIN {X 0,Y 517.395,Z 468.367,A -85,B 0,C 180,E1 -5101.613,E2 -5101.613} C_VEL
LIN {X 0,Y 517.282,Z 473.739,A -85,B 0,C 180,E1 -5103.362,E2 -5103.362} C_VEL
LIN {X 0,Y 517.046,Z 482.305,A -85,B 0,C 180,E1 -5106.36,E2 -5106.36} C_VEL
LIN {X 0,Y 516.911,Z 490.871,A -85,B 0,C 180,E1 -5109.298,E2 -5109.298} C_VEL
LIN {X 0,Y 516.704,Z 500.661,A -85,B 0,C 180,E1 -5112.588,E2 -5112.588} C_VEL
LIN {X 0,Y 516.676,Z 502.599,A -85,B 0,C 180,E1 -5113.199,E2 -5113.199} C_VEL
LIN {X 0,Y 519.564,Z 516.699,A -85,B 0,C 180,E1 -5113.578,E2 -5113.578} C_VEL
LIN {X 0,Y 519.233,Z 530.77,A -85,B 0,C 180,E1 -5114.011,E2 -5114.011} C_VEL
LIN {X 0,Y 518.905,Z 544.18,A -85,B 0,C 180,E1 -5114.586,E2 -5114.586} C_VEL
LIN {X 0,Y 518.536,Z 556.679,A -85,B 0,C 180,E1 -5115.278,E2 -5115.278} C_VEL
LIN {X 0,Y 518.069,Z 569.462,A -85,B 0,C 180,E1 -5116.167,E2 -5116.167} C_VEL
LIN {X 0,Y 517.673,Z 580.964,A -85,B 0,C 180,E1 -5117.155,E2 -5117.155} C_VEL
LIN {X 0,Y 517.335,Z 591.382,A -85,B 0,C 180,E1 -5118.242,E2 -5118.242} C_VEL
LIN {X 0,Y 516.994,Z 600.799,A -85,B 0,C 180,E1 -5119.425,E2 -5119.425} C_VEL
LIN {X 0,Y 516.71,Z 609.811,A -85,B 0,C 180,E1 -5120.804,E2 -5120.804} C_VEL
LIN {X 0,Y 516.501,Z 617.069,A -85,B 0,C 180,E1 -5122.18,E2 -5122.18} C_VEL
LIN {X 0,Y 516.385,Z 623.582,A -85,B 0,C 180,E1 -5123.749,E2 -5123.749} C_VEL
LIN {X 0,Y 516.306,Z 627.395,A -85,B 0,C 180,E1 -5124.924,E2 -5124.924} C_VEL
LIN {X 0,Y 516.324,Z 630.313,A -85,B 0,C 180,E1 -5126.098,E2 -5126.098} C_VEL
LIN {X 0,Y 516.259,Z 632.997,A -85,B 0,C 180,E1 -5127.659,E2 -5127.659} C_VEL
LIN {X 0,Y 516.157,Z 634.332,A -85,B 0,C 180,E1 -5129.22,E2 -5129.22} C_VEL
LIN {X 0,Y 516.157,Z 634.331,A -85,B 0,C 180,E1 -5130.78,E2 -5130.78} C_VEL
LIN {X 0,Y 516.259,Z 632.997,A -85,B 0,C 180,E1 -5132.341,E2 -5132.341} C_VEL
LIN {X 0,Y 516.325,Z 630.317,A -85,B 0,C 180,E1 -5133.902,E2 -5133.902} C_VEL
LIN {X 0,Y 516.383,Z 626.218,A -85,B 0,C 180,E1 -5135.467,E2 -5135.467} C_VEL
LIN {X 0,Y 516.406,Z 620.548,A -85,B 0,C 180,E1 -5137.036,E2 -5137.036} C_VEL
LIN {X 0,Y 516.599,Z 614.145,A -85,B 0,C 180,E1 -5138.41,E2 -5138.41} C_VEL
LIN {X 0,Y 516.827,Z 606.169,A -85,B 0,C 180,E1 -5139.787,E2 -5139.787} C_VEL
LIN {X 0,Y 517.108,Z 597.85,A -85,B 0,C 180,E1 -5140.969,E2 -5140.969} C_VEL
LIN {X 0,Y 517.456,Z 587.432,A -85,B 0,C 180,E1 -5142.197,E2 -5142.197} C_VEL
LIN {X 0,Y 517.811,Z 576.622,A -85,B 0,C 180,E1 -5143.24,E2 -5143.24} C_VEL
LIN {X 0,Y 518.228,Z 564.103,A -85,B 0,C 180,E1 -5144.229,E2 -5144.229} C_VEL
LIN {X 0,Y 518.718,Z 551.678,A -85,B 0,C 180,E1 -5145.018,E2 -5145.018} C_VEL
LIN {X 0,Y 519.067,Z 538.889,A -85,B 0,C 180,E1 -5145.661,E2 -5145.661} C_VEL
LIN {X 0,Y 519.371,Z 524.991,A -85,B 0,C 180,E1 -5146.188,E2 -5146.188} C_VEL
LIN {X 0,Y 519.383,Z 515.619,A -85,B 0,C 180,E1 -5146.456,E2 -5146.456} C_VEL
LIN {X 0,Y 516.67,Z 502.42,A -85,B 0,C 180,E1 -5146.827,E2 -5146.827} C_VEL
LIN {X 0,Y 516.84,Z 493.319,A -85,B 0,C 180,E1 -5149.874,E2 -5149.874} C_VEL
LIN {X 0,Y 516.967,Z 484.754,A -85,B 0,C 180,E1 -5152.795,E2 -5152.795} C_VEL
LIN {X 0,Y 517.198,Z 477.41,A -85,B 0,C 180,E1 -5155.343,E2 -5155.343} C_VEL
LIN {X 0,Y 517.372,Z 469.761,A -85,B 0,C 180,E1 -5157.998,E2 -5157.998} C_VEL
LIN {X 0,Y 517.473,Z 461.882,A -85,B 0,C 180,E1 -5160.617,E2 -5160.617} C_VEL
LIN {X 0,Y 517.601,Z 453.917,A -85,B 0,C 180,E1 -5163.361,E2 -5163.361} C_VEL
LIN {X 0,Y 517.726,Z 445.874,A -85,B 0,C 180,E1 -5166.193,E2 -5166.193} C_VEL
LIN {X 0,Y 517.817,Z 439.177,A -85,B 0,C 180,E1 -5168.633,E2 -5168.633} C_VEL
LIN {X 0,Y 517.955,Z 431.029,A -85,B 0,C 180,E1 -5171.731,E2 -5171.731} C_VEL
LIN {X 0,Y 518.245,Z 423.172,A -85,B 0,C 180,E1 -5174.844,E2 -5174.844} C_VEL
LIN {X 0,Y 518.223,Z 417.774,A -85,B 0,C 180,E1 -5177.082,E2 -5177.082} C_VEL
LIN {X 0,Y 517.364,Z 412.264,A -85,B 0,C 180,E1 -5179.528,E2 -5179.528} C_VEL
LIN {X 0,Y 516.883,Z 409.727,A -85,B 0,C 180,E1 -5180.724,E2 -5180.724} C_VEL
LIN {X 0,Y 516.885,Z 409.726,A -85,B 0,C 180,E1 -5183.342,E2 -5183.342} C_VEL
LIN {X 0,Y 516.912,Z 409.721,A -85,B 0,C 180,E1 -5186.121,E2 -5186.121} C_VEL
LIN {X 0,Y 516.893,Z 409.724,A -85,B 0,C 180,E1 -5188.936,E2 -5188.936} C_VEL
LIN {X 0,Y 516.921,Z 409.722,A -85,B 0,C 180,E1 -5191.585,E2 -5191.585} C_VEL
LIN {X 0,Y 516.934,Z 409.715,A -85,B 0,C 180,E1 -5194.211,E2 -5194.211} C_VEL
LIN {X 0,Y 516.875,Z 409.725,A -85,B 0,C 180,E1 -5196.777,E2 -5196.777} C_VEL
LIN {X 0,Y 516.942,Z 409.711,A -85,B 0,C 180,E1 -5199.732,E2 -5199.732} C_VEL
LIN {X 0,Y 516.932,Z 409.718,A -85,B 0,C 180,E1 -5202.596,E2 -5202.596} C_VEL
LIN {X 0,Y 516.945,Z 409.714,A -85,B 0,C 180,E1 -5205.03,E2 -5205.03} C_VEL
LIN {X 0,Y 516.968,Z 409.715,A -85,B 0,C 180,E1 -5208.234,E2 -5208.234} C_VEL
LIN {X 0,Y 516.961,Z 409.711,A -85,B 0,C 180,E1 -5211.4,E2 -5211.4} C_VEL
LIN {X 0,Y 517.014,Z 409.71,A -85,B 0,C 180,E1 -5213.757,E2 -5213.757} C_VEL
LIN {X 0,Y 517.085,Z 409.694,A -85,B 0,C 180,E1 -5217.663,E2 -5217.663} C_VEL
LIN {X 0,Y 517.096,Z 409.697,A -85,B 0,C 180,E1 -5220.779,E2 -5220.779} C_VEL
LIN {X 0,Y 517.015,Z 409.706,A -85,B 0,C 180,E1 -5223.117,E2 -5223.117} C_VEL
LIN {X 0,Y 517.012,Z 409.71,A -85,B 0,C 180,E1 -5226.243,E2 -5226.243} C_VEL
LIN {X 0,Y 516.956,Z 409.715,A -85,B 0,C 180,E1 -5229.389,E2 -5229.389} C_VEL
LIN {X 0,Y 516.955,Z 409.718,A -85,B 0,C 180,E1 -5231.807,E2 -5231.807} C_VEL
LIN {X 0,Y 516.947,Z 409.72,A -85,B 0,C 180,E1 -5235.147,E2 -5235.147} C_VEL
LIN {X 0,Y 516.928,Z 409.718,A -85,B 0,C 180,E1 -5238.222,E2 -5238.222} C_VEL
LIN {X 0,Y 516.915,Z 409.722,A -85,B 0,C 180,E1 -5240.701,E2 -5240.701} C_VEL
LIN {X 0,Y 516.893,Z 409.726,A -85,B 0,C 180,E1 -5244.073,E2 -5244.073} C_VEL
LIN {X 0,Y 516.929,Z 409.717,A -85,B 0,C 180,E1 -5246.658,E2 -5246.658} C_VEL
LIN {X 0,Y 516.913,Z 409.72,A -85,B 0,C 180,E1 -5249.524,E2 -5249.524} C_VEL
LIN {X 0,Y 516.898,Z 409.722,A -85,B 0,C 180,E1 -5252.543,E2 -5252.543} C_VEL
LIN {X 0,Y 516.868,Z 409.725,A -85,B 0,C 180,E1 -5255.33,E2 -5255.33} C_VEL
LIN {X 0,Y 516.883,Z 409.726,A -85,B 0,C 180,E1 -5257.943,E2 -5257.943} C_VEL
LIN {X 0,Y 516.886,Z 409.728,A -85,B 0,C 180,E1 -5260.742,E2 -5260.742} C_VEL
LIN {X 0,Y 516.907,Z 409.722,A -85,B 0,C 180,E1 -5262.829,E2 -5262.829} C_VEL
LIN {X 0,Y 516.925,Z 409.723,A -85,B 0,C 180,E1 -5265.01,E2 -5265.01} C_VEL
LIN {X 0,Y 516.917,Z 409.727,A -85,B 0,C 180,E1 -5268.399,E2 -5268.399} C_VEL
LIN {X 0,Y 516.884,Z 409.729,A -85,B 0,C 180,E1 -5269.12,E2 -5269.12} C_VEL
LIN {X 0,Y 516.318,Z 410.273,A -85,B 0,C 180,E1 -5269.767,E2 -5269.767} C_VEL
LIN {X 0,Y 514.976,Z 411.664,A -85,B 0,C 180,E1 -5270.39,E2 -5270.39} C_VEL
LIN {X 0,Y 511.832,Z 415.908,A -85,B 0,C 180,E1 -5271.598,E2 -5271.598} C_VEL
LIN {X 0,Y 510.96,Z 418.275,A -85,B 0,C 180,E1 -5272.212,E2 -5272.212} C_VEL
LIN {X 0,Y 510.894,Z 419.034,A -85,B 0,C 180,E1 -5272.42,E2 -5272.42} C_VEL
LIN {X 0,Y 510.653,Z 428.813,A -85,B 0,C 180,E1 -5275.169,E2 -5275.169} C_VEL
LIN {X 0,Y 510.559,Z 440.208,A -85,B 0,C 180,E1 -5278.461,E2 -5278.461} C_VEL
LIN {X 0,Y 510.43,Z 449.597,A -85,B 0,C 180,E1 -5281.19,E2 -5281.19} C_VEL
LIN {X 0,Y 510.294,Z 458.854,A -85,B 0,C 180,E1 -5283.85,E2 -5283.85} C_VEL
LIN {X 0,Y 510.113,Z 471.181,A -85,B 0,C 180,E1 -5287.309,E2 -5287.309} C_VEL
LIN {X 0,Y 509.934,Z 481.811,A -85,B 0,C 180,E1 -5290.265,E2 -5290.265} C_VEL
LIN {X 0,Y 509.739,Z 491.598,A -85,B 0,C 180,E1 -5292.989,E2 -5292.989} C_VEL
LIN {X 0,Y 512.74,Z 506.758,A -85,B 0,C 180,E1 -5293.402,E2 -5293.402} C_VEL
LIN {X 0,Y 512.433,Z 520.523,A -85,B 0,C 180,E1 -5293.828,E2 -5293.828} C_VEL
LIN {X 0,Y 512.127,Z 533.339,A -85,B 0,C 180,E1 -5294.376,E2 -5294.376} C_VEL
LIN {X 0,Y 511.69,Z 546.05,A -85,B 0,C 180,E1 -5295.076,E2 -5295.076} C_VEL
LIN {X 0,Y 511.241,Z 557.676,A -85,B 0,C 180,E1 -5295.877,E2 -5295.877} C_VEL
LIN {X 0,Y 510.781,Z 569.495,A -85,B 0,C 180,E1 -5296.878,E2 -5296.878} C_VEL
LIN {X 0,Y 510.353,Z 580.044,A -85,B 0,C 180,E1 -5297.963,E2 -5297.963} C_VEL
LIN {X 0,Y 510.092,Z 589.074,A -85,B 0,C 180,E1 -5299.08,E2 -5299.08} C_VEL
LIN {X 0,Y 509.764,Z 597.192,A -85,B 0,C 180,E1 -5300.277,E2 -5300.277} C_VEL
LIN {X 0,Y 509.528,Z 604.952,A -85,B 0,C 180,E1 -5301.673,E2 -5301.673} C_VEL
LIN {X 0,Y 509.331,Z 610.391,A -85,B 0,C 180,E1 -5302.866,E2 -5302.866} C_VEL
LIN {X 0,Y 509.322,Z 616.087,A -85,B 0,C 180,E1 -5304.457,E2 -5304.457} C_VEL
LIN {X 0,Y 509.22,Z 620.238,A -85,B 0,C 180,E1 -5306.043,E2 -5306.043} C_VEL
LIN {X 0,Y 509.16,Z 622.963,A -85,B 0,C 180,E1 -5307.627,E2 -5307.627} C_VEL
LIN {X 0,Y 509.07,Z 624.315,A -85,B 0,C 180,E1 -5309.209,E2 -5309.209} C_VEL
LIN {X 0,Y 509.071,Z 624.36,A -85,B 0,C 180,E1 -5310.791,E2 -5310.791} C_VEL
LIN {X 0,Y 509.159,Z 623.07,A -85,B 0,C 180,E1 -5312.373,E2 -5312.373} C_VEL
LIN {X 0,Y 509.22,Z 620.433,A -85,B 0,C 180,E1 -5313.957,E2 -5313.957} C_VEL
LIN {X 0,Y 509.318,Z 616.364,A -85,B 0,C 180,E1 -5315.543,E2 -5315.543} C_VEL
LIN {X 0,Y 509.33,Z 610.751,A -85,B 0,C 180,E1 -5317.134,E2 -5317.134} C_VEL
LIN {X 0,Y 509.509,Z 605.398,A -85,B 0,C 180,E1 -5318.328,E2 -5318.328} C_VEL
LIN {X 0,Y 509.732,Z 597.735,A -85,B 0,C 180,E1 -5319.724,E2 -5319.724} C_VEL
LIN {X 0,Y 510.057,Z 589.727,A -85,B 0,C 180,E1 -5320.921,E2 -5320.921} C_VEL
LIN {X 0,Y 510.434,Z 579.78,A -85,B 0,C 180,E1 -5322.156,E2 -5322.156} C_VEL
LIN {X 0,Y 510.846,Z 568.324,A -85,B 0,C 180,E1 -5323.323,E2 -5323.323} C_VEL
LIN {X 0,Y 511.308,Z 556.15,A -85,B 0,C 180,E1 -5324.324,E2 -5324.324} C_VEL
LIN {X 0,Y 511.727,Z 544.159,A -85,B 0,C 180,E1 -5325.126,E2 -5325.126} C_VEL
LIN {X 0,Y 512.159,Z 530.932,A -85,B 0,C 180,E1 -5325.827,E2 -5325.827} C_VEL
LIN {X 0,Y 512.542,Z 516.98,A -85,B 0,C 180,E1 -5326.385,E2 -5326.385} C_VEL
LIN {X 0,Y 512.56,Z 505.54,A -85,B 0,C 180,E1 -5326.724,E2 -5326.724} C_VEL
LIN {X 0,Y 509.758,Z 491.538,A -85,B 0,C 180,E1 -5327.113,E2 -5327.113} C_VEL
LIN {X 0,Y 509.962,Z 480.644,A -85,B 0,C 180,E1 -5330.153,E2 -5330.153} C_VEL
LIN {X 0,Y 510.105,Z 469.972,A -85,B 0,C 180,E1 -5333.12,E2 -5333.12} C_VEL
LIN {X 0,Y 510.312,Z 458.048,A -85,B 0,C 180,E1 -5336.468,E2 -5336.468} C_VEL
LIN {X 0,Y 510.449,Z 448.358,A -85,B 0,C 180,E1 -5339.26,E2 -5339.26} C_VEL
LIN {X 0,Y 510.584,Z 438.93,A -85,B 0,C 180,E1 -5342.001,E2 -5342.001} C_VEL
LIN {X 0,Y 510.687,Z 427.451,A -85,B 0,C 180,E1 -5345.31,E2 -5345.31} C_VEL
LIN {X 0,Y 510.894,Z 418.775,A -85,B 0,C 180,E1 -5347.745,E2 -5347.745} C_VEL
LIN {X 0,Y 510.646,Z 415.058,A -85,B 0,C 180,E1 -5348.782,E2 -5348.782} C_VEL
LIN {X 0,Y 509.876,Z 410.602,A -85,B 0,C 180,E1 -5350.091,E2 -5350.091} C_VEL
LIN {X 0,Y 509.827,Z 410.607,A -85,B 0,C 180,E1 -5353.062,E2 -5353.062} C_VEL
LIN {X 0,Y 509.833,Z 410.608,A -85,B 0,C 180,E1 -5355.792,E2 -5355.792} C_VEL
LIN {X 0,Y 509.86,Z 410.604,A -85,B 0,C 180,E1 -5358.575,E2 -5358.575} C_VEL
LIN {X 0,Y 509.853,Z 410.606,A -85,B 0,C 180,E1 -5361.786,E2 -5361.786} C_VEL
LIN {X 0,Y 509.846,Z 410.603,A -85,B 0,C 180,E1 -5364.623,E2 -5364.623} C_VEL
LIN {X 0,Y 509.863,Z 410.601,A -85,B 0,C 180,E1 -5367.481,E2 -5367.481} C_VEL
LIN {X 0,Y 509.884,Z 410.596,A -85,B 0,C 180,E1 -5370.269,E2 -5370.269} C_VEL
LIN {X 0,Y 509.886,Z 410.598,A -85,B 0,C 180,E1 -5372.944,E2 -5372.944} C_VEL
LIN {X 0,Y 509.873,Z 410.598,A -85,B 0,C 180,E1 -5375.574,E2 -5375.574} C_VEL
LIN {X 0,Y 509.825,Z 410.605,A -85,B 0,C 180,E1 -5378.149,E2 -5378.149} C_VEL
LIN {X 0,Y 509.868,Z 410.601,A -85,B 0,C 180,E1 -5380.682,E2 -5380.682} C_VEL
LIN {X 0,Y 509.882,Z 410.601,A -85,B 0,C 180,E1 -5380.957,E2 -5380.957} C_VEL
LIN {X 0,Y 513.302,Z 422.102,A -85,B 0,C 180,E1 -5381.531,E2 -5381.531} C_VEL
LIN {X 0,Y 512.846,Z 437.18,A -85,B 0,C 180,E1 -5382.257,E2 -5382.257} C_VEL
LIN {X 0,Y 512.345,Z 450.196,A -85,B 0,C 180,E1 -5383.053,E2 -5383.053} C_VEL
LIN {X 0,Y 511.87,Z 461.156,A -85,B 0,C 180,E1 -5383.857,E2 -5383.857} C_VEL
LIN {X 0,Y 511.329,Z 472.638,A -85,B 0,C 180,E1 -5384.862,E2 -5384.862} C_VEL
LIN {X 0,Y 510.897,Z 482.457,A -85,B 0,C 180,E1 -5385.867,E2 -5385.867} C_VEL
LIN {X 0,Y 510.463,Z 492.473,A -85,B 0,C 180,E1 -5387.072,E2 -5387.072} C_VEL
LIN {X 0,Y 510.058,Z 502.405,A -85,B 0,C 180,E1 -5388.516,E2 -5388.516} C_VEL
LIN {X 0,Y 509.779,Z 509.136,A -85,B 0,C 180,E1 -5389.675,E2 -5389.675} C_VEL
LIN {X 0,Y 509.588,Z 515.06,A -85,B 0,C 180,E1 -5390.874,E2 -5390.874} C_VEL
LIN {X 0,Y 509.469,Z 520.07,A -85,B 0,C 180,E1 -5392.071,E2 -5392.071} C_VEL
LIN {X 0,Y 509.308,Z 524.91,A -85,B 0,C 180,E1 -5393.482,E2 -5393.482} C_VEL
LIN {X 0,Y 509.305,Z 527.681,A -85,B 0,C 180,E1 -5394.457,E2 -5394.457} C_VEL
LIN {X 0,Y 509.236,Z 531.09,A -85,B 0,C 180,E1 -5396.043,E2 -5396.043} C_VEL
LIN {X 0,Y 509.189,Z 532.439,A -85,B 0,C 180,E1 -5396.835,E2 -5396.835} C_VEL
LIN {X 0,Y 509.109,Z 534.109,A -85,B 0,C 180,E1 -5398.418,E2 -5398.418} C_VEL
LIN {X 0,Y 509.063,Z 534.666,A -85,B 0,C 180,E1 -5400,E2 -5400} C_VEL
LIN {X 0,Y 509.072,Z 534.614,A -85,B 0,C 180,E1 -5400.791,E2 -5400.791} C_VEL
LIN {X 0,Y 509.187,Z 533.519,A -85,B 0,C 180,E1 -5402.373,E2 -5402.373} C_VEL
LIN {X 0,Y 509.236,Z 531.292,A -85,B 0,C 180,E1 -5403.957,E2 -5403.957} C_VEL
LIN {X 0,Y 509.166,Z 529.837,A -85,B 0,C 180,E1 -5404.75,E2 -5404.75} C_VEL
LIN {X 0,Y 509.324,Z 525.831,A -85,B 0,C 180,E1 -5406.338,E2 -5406.338} C_VEL
LIN {X 0,Y 509.459,Z 520.505,A -85,B 0,C 180,E1 -5407.929,E2 -5407.929} C_VEL
LIN {X 0,Y 509.594,Z 515.591,A -85,B 0,C 180,E1 -5409.126,E2 -5409.126} C_VEL
LIN {X 0,Y 509.885,Z 508.697,A -85,B 0,C 180,E1 -5410.523,E2 -5410.523} C_VEL
LIN {X 0,Y 510.217,Z 499.616,A -85,B 0,C 180,E1 -5412.042,E2 -5412.042} C_VEL
LIN {X 0,Y 510.627,Z 490.247,A -85,B 0,C 180,E1 -5413.329,E2 -5413.329} C_VEL
LIN {X 0,Y 511.059,Z 479.804,A -85,B 0,C 180,E1 -5414.535,E2 -5414.535} C_VEL
LIN {X 0,Y 511.555,Z 468.633,A -85,B 0,C 180,E1 -5415.62,E2 -5415.62} C_VEL
LIN {X 0,Y 512.106,Z 455.94,A -85,B 0,C 180,E1 -5416.637,E2 -5416.637} C_VEL
LIN {X 0,Y 512.571,Z 443.588,A -85,B 0,C 180,E1 -5417.454,E2 -5417.454} C_VEL
LIN {X 0,Y 513.037,Z 429.407,A -85,B 0,C 180,E1 -5418.21,E2 -5418.21} C_VEL
LIN {X 0,Y 513.028,Z 420.713,A -85,B 0,C 180,E1 -5418.594,E2 -5418.594} C_VEL
LIN {X 0,Y 509.872,Z 410.598,A -85,B 0,C 180,E1 -5419.083,E2 -5419.083} C_VEL
LIN {X 0,Y 509.853,Z 410.599,A -85,B 0,C 180,E1 -5421.002,E2 -5421.002} C_VEL
LIN {X 0,Y 509.826,Z 410.605,A -85,B 0,C 180,E1 -5423.564,E2 -5423.564} C_VEL
LIN {X 0,Y 509.914,Z 410.594,A -85,B 0,C 180,E1 -5426.379,E2 -5426.379} C_VEL
LIN {X 0,Y 509.879,Z 410.596,A -85,B 0,C 180,E1 -5428.844,E2 -5428.844} C_VEL
LIN {X 0,Y 509.828,Z 410.606,A -85,B 0,C 180,E1 -5431.59,E2 -5431.59} C_VEL
LIN {X 0,Y 509.849,Z 410.599,A -85,B 0,C 180,E1 -5434.414,E2 -5434.414} C_VEL
LIN {X 0,Y 509.818,Z 410.606,A -85,B 0,C 180,E1 -5437.341,E2 -5437.341} C_VEL
LIN {X 0,Y 509.84,Z 410.601,A -85,B 0,C 180,E1 -5440.382,E2 -5440.382} C_VEL
LIN {X 0,Y 509.843,Z 410.604,A -85,B 0,C 180,E1 -5443.064,E2 -5443.064} C_VEL
LIN {X 0,Y 509.936,Z 410.687,A -85,B 0,C 180,E1 -5444.594,E2 -5444.594} C_VEL
LIN {X 0,Y 509.697,Z 418.105,A -85,B 0,C 180,E1 -5446.953,E2 -5446.953} C_VEL
LIN {X 0,Y 509.895,Z 430.425,A -85,B 0,C 180,E1 -5450.652,E2 -5450.652} C_VEL
LIN {X 0,Y 510.14,Z 440.813,A -85,B 0,C 180,E1 -5453.673,E2 -5453.673} C_VEL
LIN {X 0,Y 510.26,Z 450.892,A -85,B 0,C 180,E1 -5456.569,E2 -5456.569} C_VEL
LIN {X 0,Y 510.288,Z 460.669,A -85,B 0,C 180,E1 -5459.364,E2 -5459.364} C_VEL
LIN {X 0,Y 510.306,Z 469.192,A -85,B 0,C 180,E1 -5461.814,E2 -5461.814} C_VEL
LIN {X 0,Y 510.192,Z 477.407,A -85,B 0,C 180,E1 -5464.283,E2 -5464.283} C_VEL
LIN {X 0,Y 509.947,Z 486.333,A -85,B 0,C 180,E1 -5467.426,E2 -5467.426} C_VEL
LIN {X 0,Y 509.785,Z 494.542,A -85,B 0,C 180,E1 -5470.259,E2 -5470.259} C_VEL
LIN {X 0,Y 509.645,Z 502.599,A -85,B 0,C 180,E1 -5472.96,E2 -5472.96} C_VEL
LIN {X 0,Y 512.744,Z 517.696,A -85,B 0,C 180,E1 -5473.38,E2 -5473.38} C_VEL
LIN {X 0,Y 512.424,Z 530.527,A -85,B 0,C 180,E1 -5473.784,E2 -5473.784} C_VEL
LIN {X 0,Y 512.029,Z 544.176,A -85,B 0,C 180,E1 -5474.373,E2 -5474.373} C_VEL
LIN {X 0,Y 511.657,Z 556.677,A -85,B 0,C 180,E1 -5475.075,E2 -5475.075} C_VEL
LIN {X 0,Y 511.12,Z 569.465,A -85,B 0,C 180,E1 -5475.975,E2 -5475.975} C_VEL
LIN {X 0,Y 510.721,Z 580.961,A -85,B 0,C 180,E1 -5476.977,E2 -5476.977} C_VEL
LIN {X 0,Y 510.355,Z 591.38,A -85,B 0,C 180,E1 -5478.079,E2 -5478.079} C_VEL
LIN {X 0,Y 509.997,Z 600.797,A -85,B 0,C 180,E1 -5479.278,E2 -5479.278} C_VEL
LIN {X 0,Y 509.673,Z 609.81,A -85,B 0,C 180,E1 -5480.676,E2 -5480.676} C_VEL
LIN {X 0,Y 509.45,Z 617.071,A -85,B 0,C 180,E1 -5482.071,E2 -5482.071} C_VEL
LIN {X 0,Y 509.307,Z 623.581,A -85,B 0,C 180,E1 -5483.662,E2 -5483.662} C_VEL
LIN {X 0,Y 509.239,Z 627.395,A -85,B 0,C 180,E1 -5484.853,E2 -5484.853} C_VEL
LIN {X 0,Y 509.219,Z 630.313,A -85,B 0,C 180,E1 -5486.043,E2 -5486.043} C_VEL
LIN {X 0,Y 509.159,Z 632.997,A -85,B 0,C 180,E1 -5487.627,E2 -5487.627} C_VEL
LIN {X 0,Y 509.071,Z 634.332,A -85,B 0,C 180,E1 -5489.209,E2 -5489.209} C_VEL
LIN {X 0,Y 509.071,Z 634.33,A -85,B 0,C 180,E1 -5490.791,E2 -5490.791} C_VEL
LIN {X 0,Y 509.159,Z 632.996,A -85,B 0,C 180,E1 -5492.373,E2 -5492.373} C_VEL
LIN {X 0,Y 509.219,Z 630.316,A -85,B 0,C 180,E1 -5493.957,E2 -5493.957} C_VEL
LIN {X 0,Y 509.295,Z 626.218,A -85,B 0,C 180,E1 -5495.543,E2 -5495.543} C_VEL
LIN {X 0,Y 509.33,Z 620.55,A -85,B 0,C 180,E1 -5497.134,E2 -5497.134} C_VEL
LIN {X 0,Y 509.553,Z 614.143,A -85,B 0,C 180,E1 -5498.527,E2 -5498.527} C_VEL
LIN {X 0,Y 509.788,Z 606.168,A -85,B 0,C 180,E1 -5499.923,E2 -5499.923} C_VEL
LIN {X 0,Y 510.114,Z 597.85,A -85,B 0,C 180,E1 -5501.121,E2 -5501.121} C_VEL
LIN {X 0,Y 510.463,Z 587.762,A -85,B 0,C 180,E1 -5502.33,E2 -5502.33} C_VEL
LIN {X 0,Y 510.866,Z 576.622,A -85,B 0,C 180,E1 -5503.424,E2 -5503.424} C_VEL
LIN {X 0,Y 511.323,Z 564.101,A -85,B 0,C 180,E1 -5504.426,E2 -5504.426} C_VEL
LIN {X 0,Y 511.855,Z 551.68,A -85,B 0,C 180,E1 -5505.224,E2 -5505.224} C_VEL
LIN {X 0,Y 512.23,Z 538.894,A -85,B 0,C 180,E1 -5505.876,E2 -5505.876} C_VEL
LIN {X 0,Y 512.563,Z 524.938,A -85,B 0,C 180,E1 -5506.41,E2 -5506.41} C_VEL
LIN {X 0,Y 512.594,Z 516.85,A -85,B 0,C 180,E1 -5506.647,E2 -5506.647} C_VEL
LIN {X 0,Y 509.636,Z 502.42,A -85,B 0,C 180,E1 -5507.066,E2 -5507.066} C_VEL
LIN {X 0,Y 509.814,Z 492.68,A -85,B 0,C 180,E1 -5510.379,E2 -5510.379} C_VEL
LIN {X 0,Y 510.022,Z 483.529,A -85,B 0,C 180,E1 -5513.554,E2 -5513.554} C_VEL
LIN {X 0,Y 510.23,Z 475.197,A -85,B 0,C 180,E1 -5516.45,E2 -5516.45} C_VEL
LIN {X 0,Y 510.418,Z 466.696,A -85,B 0,C 180,E1 -5519.262,E2 -5519.262} C_VEL
LIN {X 0,Y 510.556,Z 457.439,A -85,B 0,C 180,E1 -5522.47,E2 -5522.47} C_VEL
LIN {X 0,Y 510.705,Z 448.303,A -85,B 0,C 180,E1 -5525.716,E2 -5525.716} C_VEL
LIN {X 0,Y 510.812,Z 440.046,A -85,B 0,C 180,E1 -5528.765,E2 -5528.765} C_VEL
LIN {X 0,Y 510.947,Z 433.409,A -85,B 0,C 180,E1 -5531.318,E2 -5531.318} C_VEL
LIN {X 0,Y 511.241,Z 425.406,A -85,B 0,C 180,E1 -5534.515,E2 -5534.515} C_VEL
LIN {X 0,Y 511.304,Z 420.009,A -85,B 0,C 180,E1 -5536.761,E2 -5536.761} C_VEL
LIN {X 0,Y 510.801,Z 415.676,A -85,B 0,C 180,E1 -5538.668,E2 -5538.668} C_VEL
LIN {X 0,Y 509.852,Z 410.604,A -85,B 0,C 180,E1 -5541.03,E2 -5541.03} C_VEL
LIN {X 0,Y 509.841,Z 410.602,A -85,B 0,C 180,E1 -5544.419,E2 -5544.419} C_VEL
LIN {X 0,Y 509.863,Z 410.6,A -85,B 0,C 180,E1 -5547.481,E2 -5547.481} C_VEL
LIN {X 0,Y 509.86,Z 410.601,A -85,B 0,C 180,E1 -5550.274,E2 -5550.274} C_VEL
LIN {X 0,Y 509.887,Z 410.595,A -85,B 0,C 180,E1 -5552.945,E2 -5552.945} C_VEL
LIN {X 0,Y 509.872,Z 410.597,A -85,B 0,C 180,E1 -5555.574,E2 -5555.574} C_VEL
LIN {X 0,Y 509.825,Z 410.601,A -85,B 0,C 180,E1 -5558.149,E2 -5558.149} C_VEL
LIN {X 0,Y 509.867,Z 410.599,A -85,B 0,C 180,E1 -5560.682,E2 -5560.682} C_VEL
LIN {X 0,Y 509.888,Z 410.597,A -85,B 0,C 180,E1 -5563.175,E2 -5563.175} C_VEL
LIN {X 0,Y 509.866,Z 410.593,A -85,B 0,C 180,E1 -5565.634,E2 -5565.634} C_VEL
LIN {X 0,Y 509.915,Z 410.592,A -85,B 0,C 180,E1 -5568.875,E2 -5568.875} C_VEL
LIN {X 0,Y 509.924,Z 410.587,A -85,B 0,C 180,E1 -5572.078,E2 -5572.078} C_VEL
LIN {X 0,Y 509.986,Z 410.584,A -85,B 0,C 180,E1 -5574.464,E2 -5574.464} C_VEL
LIN {X 0,Y 510.056,Z 410.57,A -85,B 0,C 180,E1 -5577.631,E2 -5577.631} C_VEL
LIN {X 0,Y 510.066,Z 410.573,A -85,B 0,C 180,E1 -5580.79,E2 -5580.79} C_VEL
LIN {X 0,Y 509.957,Z 410.585,A -85,B 0,C 180,E1 -5583.16,E2 -5583.16} C_VEL
LIN {X 0,Y 509.981,Z 410.585,A -85,B 0,C 180,E1 -5586.33,E2 -5586.33} C_VEL
LIN {X 0,Y 509.919,Z 410.588,A -85,B 0,C 180,E1 -5588.72,E2 -5588.72} C_VEL
LIN {X 0,Y 509.907,Z 410.597,A -85,B 0,C 180,E1 -5591.932,E2 -5591.932} C_VEL
LIN {X 0,Y 509.896,Z 410.597,A -85,B 0,C 180,E1 -5595.242,E2 -5595.242} C_VEL
LIN {X 0,Y 509.891,Z 410.596,A -85,B 0,C 180,E1 -5598.001,E2 -5598.001} C_VEL
LIN {X 0,Y 509.853,Z 410.605,A -85,B 0,C 180,E1 -5601.002,E2 -5601.002} C_VEL
LIN {X 0,Y 509.825,Z 410.601,A -85,B 0,C 180,E1 -5603.564,E2 -5603.564} C_VEL
LIN {X 0,Y 509.914,Z 410.59,A -85,B 0,C 180,E1 -5606.379,E2 -5606.379} C_VEL
LIN {X 0,Y 509.879,Z 410.598,A -85,B 0,C 180,E1 -5608.844,E2 -5608.844} C_VEL
LIN {X 0,Y 509.823,Z 410.609,A -85,B 0,C 180,E1 -5611.59,E2 -5611.59} C_VEL
LIN {X 0,Y 509.849,Z 410.603,A -85,B 0,C 180,E1 -5614.414,E2 -5614.414} C_VEL
LIN {X 0,Y 509.819,Z 410.607,A -85,B 0,C 180,E1 -5617.341,E2 -5617.341} C_VEL
LIN {X 0,Y 509.84,Z 410.604,A -85,B 0,C 180,E1 -5620.382,E2 -5620.382} C_VEL
LIN {X 0,Y 509.842,Z 410.602,A -85,B 0,C 180,E1 -5623.064,E2 -5623.064} C_VEL
LIN {X 0,Y 509.833,Z 410.605,A -85,B 0,C 180,E1 -5625.792,E2 -5625.792} C_VEL
LIN {X 0,Y 509.859,Z 410.606,A -85,B 0,C 180,E1 -5628.575,E2 -5628.575} C_VEL
LIN {X 0,Y 509.899,Z 410.748,A -85,B 0,C 180,E1 -5630.089,E2 -5630.089} C_VEL
LIN {X 0,Y 510.862,Z 416.626,A -85,B 0,C 180,E1 -5631.752,E2 -5631.752} C_VEL
LIN {X 0,Y 510.894,Z 419.034,A -85,B 0,C 180,E1 -5632.42,E2 -5632.42} C_VEL
LIN {X 0,Y 510.232,Z 421.334,A -85,B 0,C 180,E1 -5633.025,E2 -5633.025} C_VEL
LIN {X 0,Y 507.329,Z 425.337,A -85,B 0,C 180,E1 -5633.993,E2 -5633.993} C_VEL
LIN {X 0,Y 504.376,Z 429.329,A -85,B 0,C 180,E1 -5634.971,E2 -5634.971} C_VEL
LIN {X 0,Y 503.655,Z 431.581,A -85,B 0,C 180,E1 -5635.59,E2 -5635.59} C_VEL
LIN {X 0,Y 503.569,Z 442.951,A -85,B 0,C 180,E1 -5638.91,E2 -5638.91} C_VEL
LIN {X 0,Y 503.426,Z 453.895,A -85,B 0,C 180,E1 -5642.117,E2 -5642.117} C_VEL
LIN {X 0,Y 503.13,Z 464.667,A -85,B 0,C 180,E1 -5645.225,E2 -5645.225} C_VEL
LIN {X 0,Y 503.019,Z 473.97,A -85,B 0,C 180,E1 -5647.837,E2 -5647.837} C_VEL
LIN {X 0,Y 502.849,Z 484.682,A -85,B 0,C 180,E1 -5650.826,E2 -5650.826} C_VEL
LIN {X 0,Y 502.73,Z 491.555,A -85,B 0,C 180,E1 -5652.745,E2 -5652.745} C_VEL
LIN {X 0,Y 505.867,Z 507.019,A -85,B 0,C 180,E1 -5653.176,E2 -5653.176} C_VEL
LIN {X 0,Y 505.594,Z 521.153,A -85,B 0,C 180,E1 -5653.625,E2 -5653.625} C_VEL
LIN {X 0,Y 505.299,Z 533.372,A -85,B 0,C 180,E1 -5654.16,E2 -5654.16} C_VEL
LIN {X 0,Y 504.829,Z 546.09,A -85,B 0,C 180,E1 -5654.869,E2 -5654.869} C_VEL
LIN {X 0,Y 504.306,Z 557.721,A -85,B 0,C 180,E1 -5655.678,E2 -5655.678} C_VEL
LIN {X 0,Y 503.834,Z 569.543,A -85,B 0,C 180,E1 -5656.694,E2 -5656.694} C_VEL
LIN {X 0,Y 503.422,Z 579.724,A -85,B 0,C 180,E1 -5657.751,E2 -5657.751} C_VEL
LIN {X 0,Y 503.096,Z 589.127,A -85,B 0,C 180,E1 -5658.926,E2 -5658.926} C_VEL
LIN {X 0,Y 502.726,Z 597.246,A -85,B 0,C 180,E1 -5660.139,E2 -5660.139} C_VEL
LIN {X 0,Y 502.472,Z 605.008,A -85,B 0,C 180,E1 -5661.555,E2 -5661.555} C_VEL
LIN {X 0,Y 502.256,Z 610.449,A -85,B 0,C 180,E1 -5662.765,E2 -5662.765} C_VEL
LIN {X 0,Y 502.234,Z 616.145,A -85,B 0,C 180,E1 -5664.379,E2 -5664.379} C_VEL
LIN {X 0,Y 502.117,Z 620.293,A -85,B 0,C 180,E1 -5665.987,E2 -5665.987} C_VEL
LIN {X 0,Y 502.064,Z 623.01,A -85,B 0,C 180,E1 -5667.593,E2 -5667.593} C_VEL
LIN {X 0,Y 501.987,Z 624.378,A -85,B 0,C 180,E1 -5669.198,E2 -5669.198} C_VEL
LIN {X 0,Y 501.988,Z 624.421,A -85,B 0,C 180,E1 -5670.802,E2 -5670.802} C_VEL
LIN {X 0,Y 502.064,Z 623.131,A -85,B 0,C 180,E1 -5672.407,E2 -5672.407} C_VEL
LIN {X 0,Y 502.117,Z 620.485,A -85,B 0,C 180,E1 -5674.013,E2 -5674.013} C_VEL
LIN {X 0,Y 502.23,Z 616.418,A -85,B 0,C 180,E1 -5675.621,E2 -5675.621} C_VEL
LIN {X 0,Y 502.255,Z 610.804,A -85,B 0,C 180,E1 -5677.235,E2 -5677.235} C_VEL
LIN {X 0,Y 502.444,Z 605.448,A -85,B 0,C 180,E1 -5678.446,E2 -5678.446} C_VEL
LIN {X 0,Y 502.696,Z 597.782,A -85,B 0,C 180,E1 -5679.861,E2 -5679.861} C_VEL
LIN {X 0,Y 503.048,Z 589.77,A -85,B 0,C 180,E1 -5681.075,E2 -5681.075} C_VEL
LIN {X 0,Y 503.425,Z 580.473,A -85,B 0,C 180,E1 -5682.251,E2 -5682.251} C_VEL
LIN {X 0,Y 503.867,Z 569.415,A -85,B 0,C 180,E1 -5683.408,E2 -5683.408} C_VEL
LIN {X 0,Y 504.34,Z 557.552,A -85,B 0,C 180,E1 -5684.424,E2 -5684.424} C_VEL
LIN {X 0,Y 504.82,Z 545.877,A -85,B 0,C 180,E1 -5685.235,E2 -5685.235} C_VEL
LIN {X 0,Y 505.291,Z 532.018,A -85,B 0,C 180,E1 -5685.996,E2 -5685.996} C_VEL
LIN {X 0,Y 505.707,Z 517.898,A -85,B 0,C 180,E1 -5686.58,E2 -5686.58} C_VEL
LIN {X 0,Y 505.768,Z 506.736,A -85,B 0,C 180,E1 -5686.924,E2 -5686.924} C_VEL
LIN {X 0,Y 502.744,Z 491.533,A -85,B 0,C 180,E1 -5687.347,E2 -5687.347} C_VEL
LIN {X 0,Y 502.918,Z 480.016,A -85,B 0,C 180,E1 -5690.562,E2 -5690.562} C_VEL
LIN {X 0,Y 503.038,Z 469.629,A -85,B 0,C 180,E1 -5693.464,E2 -5693.464} C_VEL
LIN {X 0,Y 503.298,Z 458.825,A -85,B 0,C 180,E1 -5696.541,E2 -5696.541} C_VEL
LIN {X 0,Y 503.45,Z 449.547,A -85,B 0,C 180,E1 -5699.248,E2 -5699.248} C_VEL
LIN {X 0,Y 503.589,Z 440.074,A -85,B 0,C 180,E1 -5702.027,E2 -5702.027} C_VEL
LIN {X 0,Y 503.687,Z 430.225,A -85,B 0,C 180,E1 -5704.895,E2 -5704.895} C_VEL
LIN {X 0,Y 503.942,Z 421.607,A -85,B 0,C 180,E1 -5707.352,E2 -5707.352} C_VEL
LIN {X 0,Y 503.783,Z 417.113,A -85,B 0,C 180,E1 -5708.627,E2 -5708.627} C_VEL
LIN {X 0,Y 502.814,Z 411.482,A -85,B 0,C 180,E1 -5710.275,E2 -5710.275} C_VEL
LIN {X 0,Y 502.775,Z 411.486,A -85,B 0,C 180,E1 -5713.374,E2 -5713.374} C_VEL
LIN {X 0,Y 502.793,Z 411.484,A -85,B 0,C 180,E1 -5715.661,E2 -5715.661} C_VEL
LIN {X 0,Y 502.832,Z 411.48,A -85,B 0,C 180,E1 -5717.864,E2 -5717.864} C_VEL
LIN {X 0,Y 502.803,Z 411.482,A -85,B 0,C 180,E1 -5721.024,E2 -5721.024} C_VEL
LIN {X 0,Y 502.786,Z 411.483,A -85,B 0,C 180,E1 -5724.167,E2 -5724.167} C_VEL
LIN {X 0,Y 502.835,Z 411.476,A -85,B 0,C 180,E1 -5726.993,E2 -5726.993} C_VEL
LIN {X 0,Y 502.833,Z 411.472,A -85,B 0,C 180,E1 -5730.062,E2 -5730.062} C_VEL
LIN {X 0,Y 502.835,Z 411.478,A -85,B 0,C 180,E1 -5732.533,E2 -5732.533} C_VEL
LIN {X 0,Y 502.831,Z 411.477,A -85,B 0,C 180,E1 -5735.298,E2 -5735.298} C_VEL
LIN {X 0,Y 502.796,Z 411.481,A -85,B 0,C 180,E1 -5737.827,E2 -5737.827} C_VEL
LIN {X 0,Y 502.824,Z 411.479,A -85,B 0,C 180,E1 -5740.719,E2 -5740.719} C_VEL
LIN {X 0,Y 506.497,Z 423.523,A -85,B 0,C 180,E1 -5741.336,E2 -5741.336} C_VEL
LIN {X 0,Y 506.075,Z 437.598,A -85,B 0,C 180,E1 -5742.028,E2 -5742.028} C_VEL
LIN {X 0,Y 505.46,Z 451.888,A -85,B 0,C 180,E1 -5742.919,E2 -5742.919} C_VEL
LIN {X 0,Y 504.84,Z 465.158,A -85,B 0,C 180,E1 -5743.937,E2 -5743.937} C_VEL
LIN {X 0,Y 504.295,Z 477.22,A -85,B 0,C 180,E1 -5745.059,E2 -5745.059} C_VEL
LIN {X 0,Y 503.823,Z 488.132,A -85,B 0,C 180,E1 -5746.282,E2 -5746.282} C_VEL
LIN {X 0,Y 503.336,Z 497.339,A -85,B 0,C 180,E1 -5747.501,E2 -5747.501} C_VEL
LIN {X 0,Y 503.038,Z 505.136,A -85,B 0,C 180,E1 -5748.72,E2 -5748.72} C_VEL
LIN {X 0,Y 502.702,Z 512.83,A -85,B 0,C 180,E1 -5750.139,E2 -5750.139} C_VEL
LIN {X 0,Y 502.493,Z 519.173,A -85,B 0,C 180,E1 -5751.555,E2 -5751.555} C_VEL
LIN {X 0,Y 502.284,Z 525.062,A -85,B 0,C 180,E1 -5753.21,E2 -5753.21} C_VEL
LIN {X 0,Y 502.277,Z 528.392,A -85,B 0,C 180,E1 -5754.379,E2 -5754.379} C_VEL
LIN {X 0,Y 502.2,Z 531.825,A -85,B 0,C 180,E1 -5755.988,E2 -5755.988} C_VEL
LIN {X 0,Y 502.129,Z 534.111,A -85,B 0,C 180,E1 -5757.593,E2 -5757.593} C_VEL
LIN {X 0,Y 502.011,Z 535.303,A -85,B 0,C 180,E1 -5759.198,E2 -5759.198} C_VEL
LIN {X 0,Y 502.014,Z 535.379,A -85,B 0,C 180,E1 -5760.802,E2 -5760.802} C_VEL
LIN {X 0,Y 502.134,Z 534.307,A -85,B 0,C 180,E1 -5762.406,E2 -5762.406} C_VEL
LIN {X 0,Y 502.201,Z 532.08,A -85,B 0,C 180,E1 -5764.012,E2 -5764.012} C_VEL
LIN {X 0,Y 502.143,Z 530.597,A -85,B 0,C 180,E1 -5764.817,E2 -5764.817} C_VEL
LIN {X 0,Y 502.322,Z 526.588,A -85,B 0,C 180,E1 -5766.426,E2 -5766.426} C_VEL
LIN {X 0,Y 502.467,Z 521.264,A -85,B 0,C 180,E1 -5768.04,E2 -5768.04} C_VEL
LIN {X 0,Y 502.685,Z 514.524,A -85,B 0,C 180,E1 -5769.658,E2 -5769.658} C_VEL
LIN {X 0,Y 503.077,Z 505.999,A -85,B 0,C 180,E1 -5771.279,E2 -5771.279} C_VEL
LIN {X 0,Y 503.424,Z 497.033,A -85,B 0,C 180,E1 -5772.681,E2 -5772.681} C_VEL
LIN {X 0,Y 503.88,Z 487.564,A -85,B 0,C 180,E1 -5773.922,E2 -5773.922} C_VEL
LIN {X 0,Y 504.368,Z 476.385,A -85,B 0,C 180,E1 -5775.145,E2 -5775.145} C_VEL
LIN {X 0,Y 504.973,Z 463.994,A -85,B 0,C 180,E1 -5776.266,E2 -5776.266} C_VEL
LIN {X 0,Y 505.469,Z 451.734,A -85,B 0,C 180,E1 -5777.185,E2 -5777.185} C_VEL
LIN {X 0,Y 505.966,Z 438.663,A -85,B 0,C 180,E1 -5777.986,E2 -5777.986} C_VEL
LIN {X 0,Y 506.362,Z 424.57,A -85,B 0,C 180,E1 -5778.674,E2 -5778.674} C_VEL
LIN {X 0,Y 506.421,Z 423.187,A -85,B 0,C 180,E1 -5778.729,E2 -5778.729} C_VEL
LIN {X 0,Y 502.824,Z 411.476,A -85,B 0,C 180,E1 -5779.308,E2 -5779.308} C_VEL
LIN {X 0,Y 502.782,Z 411.485,A -85,B 0,C 180,E1 -5782.173,E2 -5782.173} C_VEL
LIN {X 0,Y 502.798,Z 411.479,A -85,B 0,C 180,E1 -5784.793,E2 -5784.793} C_VEL
LIN {X 0,Y 502.837,Z 411.476,A -85,B 0,C 180,E1 -5787.467,E2 -5787.467} C_VEL
LIN {X 0,Y 502.811,Z 411.478,A -85,B 0,C 180,E1 -5790.211,E2 -5790.211} C_VEL
LIN {X 0,Y 502.834,Z 411.473,A -85,B 0,C 180,E1 -5793.031,E2 -5793.031} C_VEL
LIN {X 0,Y 502.775,Z 411.484,A -85,B 0,C 180,E1 -5795.951,E2 -5795.951} C_VEL
LIN {X 0,Y 502.802,Z 411.478,A -85,B 0,C 180,E1 -5798.976,E2 -5798.976} C_VEL
LIN {X 0,Y 502.831,Z 411.477,A -85,B 0,C 180,E1 -5802.136,E2 -5802.136} C_VEL
LIN {X 0,Y 502.899,Z 411.556,A -85,B 0,C 180,E1 -5804.472,E2 -5804.472} C_VEL
LIN {X 0,Y 502.802,Z 416.726,A -85,B 0,C 180,E1 -5806.19,E2 -5806.19} C_VEL
LIN {X 0,Y 502.777,Z 429.808,A -85,B 0,C 180,E1 -5810.247,E2 -5810.247} C_VEL
LIN {X 0,Y 503.017,Z 439.301,A -85,B 0,C 180,E1 -5813.074,E2 -5813.074} C_VEL
LIN {X 0,Y 503.165,Z 447.566,A -85,B 0,C 180,E1 -5815.496,E2 -5815.496} C_VEL
LIN {X 0,Y 503.215,Z 457.624,A -85,B 0,C 180,E1 -5818.423,E2 -5818.423} C_VEL
LIN {X 0,Y 503.224,Z 468.767,A -85,B 0,C 180,E1 -5821.651,E2 -5821.651} C_VEL
LIN {X 0,Y 503.072,Z 479.37,A -85,B 0,C 180,E1 -5824.78,E2 -5824.78} C_VEL
LIN {X 0,Y 502.969,Z 484.752,A -85,B 0,C 180,E1 -5826.532,E2 -5826.532} C_VEL
LIN {X 0,Y 502.765,Z 493.319,A -85,B 0,C 180,E1 -5829.545,E2 -5829.545} C_VEL
LIN {X 0,Y 502.593,Z 502.599,A -85,B 0,C 180,E1 -5832.714,E2 -5832.714} C_VEL
LIN {X 0,Y 505.797,Z 517.903,A -85,B 0,C 180,E1 -5833.151,E2 -5833.151} C_VEL
LIN {X 0,Y 505.584,Z 531.787,A -85,B 0,C 180,E1 -5833.607,E2 -5833.607} C_VEL
LIN {X 0,Y 505.166,Z 545.197,A -85,B 0,C 180,E1 -5834.207,E2 -5834.207} C_VEL
LIN {X 0,Y 504.742,Z 558.256,A -85,B 0,C 180,E1 -5834.969,E2 -5834.969} C_VEL
LIN {X 0,Y 504.166,Z 570.706,A -85,B 0,C 180,E1 -5835.88,E2 -5835.88} C_VEL
LIN {X 0,Y 503.734,Z 581.979,A -85,B 0,C 180,E1 -5836.896,E2 -5836.896} C_VEL
LIN {X 0,Y 503.291,Z 593.087,A -85,B 0,C 180,E1 -5838.114,E2 -5838.114} C_VEL
LIN {X 0,Y 502.914,Z 602.224,A -85,B 0,C 180,E1 -5839.329,E2 -5839.329} C_VEL
LIN {X 0,Y 502.592,Z 610.942,A -85,B 0,C 180,E1 -5840.746,E2 -5840.746} C_VEL
LIN {X 0,Y 502.386,Z 617.072,A -85,B 0,C 180,E1 -5841.958,E2 -5841.958} C_VEL
LIN {X 0,Y 502.226,Z 623.298,A -85,B 0,C 180,E1 -5843.491,E2 -5843.491} C_VEL
LIN {X 0,Y 502.172,Z 627.396,A -85,B 0,C 180,E1 -5844.781,E2 -5844.781} C_VEL
LIN {X 0,Y 502.115,Z 630.312,A -85,B 0,C 180,E1 -5845.987,E2 -5845.987} C_VEL
LIN {X 0,Y 502.063,Z 632.996,A -85,B 0,C 180,E1 -5847.593,E2 -5847.593} C_VEL
LIN {X 0,Y 501.988,Z 634.332,A -85,B 0,C 180,E1 -5849.198,E2 -5849.198} C_VEL
LIN {X 0,Y 501.988,Z 634.33,A -85,B 0,C 180,E1 -5850.802,E2 -5850.802} C_VEL
LIN {X 0,Y 502.063,Z 632.996,A -85,B 0,C 180,E1 -5852.407,E2 -5852.407} C_VEL
LIN {X 0,Y 502.115,Z 630.315,A -85,B 0,C 180,E1 -5854.013,E2 -5854.013} C_VEL
LIN {X 0,Y 502.212,Z 626.218,A -85,B 0,C 180,E1 -5855.622,E2 -5855.622} C_VEL
LIN {X 0,Y 502.255,Z 620.552,A -85,B 0,C 180,E1 -5857.235,E2 -5857.235} C_VEL
LIN {X 0,Y 502.501,Z 614.142,A -85,B 0,C 180,E1 -5858.647,E2 -5858.647} C_VEL
LIN {X 0,Y 502.736,Z 606.167,A -85,B 0,C 180,E1 -5860.064,E2 -5860.064} C_VEL
LIN {X 0,Y 503.127,Z 597.85,A -85,B 0,C 180,E1 -5861.278,E2 -5861.278} C_VEL
LIN {X 0,Y 503.518,Z 587.19,A -85,B 0,C 180,E1 -5862.566,E2 -5862.566} C_VEL
LIN {X 0,Y 504.011,Z 575.467,A -85,B 0,C 180,E1 -5863.713,E2 -5863.713} C_VEL
LIN {X 0,Y 504.453,Z 564.099,A -85,B 0,C 180,E1 -5864.626,E2 -5864.626} C_VEL
LIN {X 0,Y 505.006,Z 551.68,A -85,B 0,C 180,E1 -5865.436,E2 -5865.436} C_VEL
LIN {X 0,Y 505.408,Z 538.898,A -85,B 0,C 180,E1 -5866.096,E2 -5866.096} C_VEL
LIN {X 0,Y 505.753,Z 524.758,A -85,B 0,C 180,E1 -5866.643,E2 -5866.643} C_VEL
LIN {X 0,Y 505.82,Z 517.985,A -85,B 0,C 180,E1 -5866.846,E2 -5866.846} C_VEL
LIN {X 0,Y 502.684,Z 503.192,A -85,B 0,C 180,E1 -5867.273,E2 -5867.273} C_VEL
LIN {X 0,Y 502.582,Z 502.42,A -85,B 0,C 180,E1 -5867.313,E2 -5867.313} C_VEL
LIN {X 0,Y 502.769,Z 493.139,A -85,B 0,C 180,E1 -5870.517,E2 -5870.517} C_VEL
LIN {X 0,Y 502.969,Z 484.752,A -85,B 0,C 180,E1 -5873.468,E2 -5873.468} C_VEL
LIN {X 0,Y 503.151,Z 476.9,A -85,B 0,C 180,E1 -5876.103,E2 -5876.103} C_VEL
LIN {X 0,Y 503.368,Z 467.552,A -85,B 0,C 180,E1 -5879.253,E2 -5879.253} C_VEL
LIN {X 0,Y 503.516,Z 458.295,A -85,B 0,C 180,E1 -5882.505,E2 -5882.505} C_VEL
LIN {X 0,Y 503.68,Z 450.294,A -85,B 0,C 180,E1 -5885.385,E2 -5885.385} C_VEL
LIN {X 0,Y 503.784,Z 442.629,A -85,B 0,C 180,E1 -5888.25,E2 -5888.25} C_VEL
LIN {X 0,Y 503.953,Z 435.169,A -85,B 0,C 180,E1 -5891.143,E2 -5891.143} C_VEL
LIN {X 0,Y 504.295,Z 426.342,A -85,B 0,C 180,E1 -5894.704,E2 -5894.704} C_VEL
LIN {X 0,Y 504.331,Z 421.059,A -85,B 0,C 180,E1 -5896.935,E2 -5896.935} C_VEL
LIN {X 0,Y 503.709,Z 416.397,A -85,B 0,C 180,E1 -5899.022,E2 -5899.022} C_VEL
LIN {X 0,Y 502.816,Z 411.48,A -85,B 0,C 180,E1 -5901.373,E2 -5901.373} C_VEL
LIN {X 0,Y 502.785,Z 411.482,A -85,B 0,C 180,E1 -5904.168,E2 -5904.168} C_VEL
LIN {X 0,Y 502.834,Z 411.478,A -85,B 0,C 180,E1 -5906.993,E2 -5906.993} C_VEL
LIN {X 0,Y 502.816,Z 411.481,A -85,B 0,C 180,E1 -5910.065,E2 -5910.065} C_VEL
LIN {X 0,Y 502.836,Z 411.475,A -85,B 0,C 180,E1 -5912.533,E2 -5912.533} C_VEL
LIN {X 0,Y 502.831,Z 411.473,A -85,B 0,C 180,E1 -5915.299,E2 -5915.299} C_VEL
LIN {X 0,Y 502.796,Z 411.478,A -85,B 0,C 180,E1 -5917.827,E2 -5917.827} C_VEL
LIN {X 0,Y 502.828,Z 411.473,A -85,B 0,C 180,E1 -5920.4,E2 -5920.4} C_VEL
LIN {X 0,Y 502.837,Z 411.474,A -85,B 0,C 180,E1 -5922.932,E2 -5922.932} C_VEL
LIN {X 0,Y 502.847,Z 411.468,A -85,B 0,C 180,E1 -5925.429,E2 -5925.429} C_VEL
LIN {X 0,Y 502.879,Z 411.468,A -85,B 0,C 180,E1 -5928.717,E2 -5928.717} C_VEL
LIN {X 0,Y 502.883,Z 411.463,A -85,B 0,C 180,E1 -5931.966,E2 -5931.966} C_VEL
LIN {X 0,Y 502.941,Z 411.461,A -85,B 0,C 180,E1 -5934.387,E2 -5934.387} C_VEL
LIN {X 0,Y 503.026,Z 411.445,A -85,B 0,C 180,E1 -5937.598,E2 -5937.598} C_VEL
LIN {X 0,Y 503.03,Z 411.455,A -85,B 0,C 180,E1 -5940,E2 -5940} C_VEL
LIN {X 0,Y 503.026,Z 411.446,A -85,B 0,C 180,E1 -5942.402,E2 -5942.402} C_VEL
LIN {X 0,Y 502.94,Z 411.462,A -85,B 0,C 180,E1 -5945.614,E2 -5945.614} C_VEL
LIN {X 0,Y 502.905,Z 411.46,A -85,B 0,C 180,E1 -5948.033,E2 -5948.033} C_VEL
LIN {X 0,Y 502.879,Z 411.469,A -85,B 0,C 180,E1 -5951.283,E2 -5951.283} C_VEL
LIN {X 0,Y 502.847,Z 411.469,A -85,B 0,C 180,E1 -5954.571,E2 -5954.571} C_VEL
LIN {X 0,Y 502.864,Z 411.472,A -85,B 0,C 180,E1 -5957.907,E2 -5957.907} C_VEL
LIN {X 0,Y 502.831,Z 411.475,A -85,B 0,C 180,E1 -5960.536,E2 -5960.536} C_VEL
LIN {X 0,Y 502.79,Z 411.477,A -85,B 0,C 180,E1 -5963.041,E2 -5963.041} C_VEL
LIN {X 0,Y 502.824,Z 411.477,A -85,B 0,C 180,E1 -5965.677,E2 -5965.677} C_VEL
LIN {X 0,Y 502.843,Z 411.476,A -85,B 0,C 180,E1 -5968.373,E2 -5968.373} C_VEL
LIN {X 0,Y 502.795,Z 411.483,A -85,B 0,C 180,E1 -5971.499,E2 -5971.499} C_VEL
LIN {X 0,Y 502.806,Z 411.478,A -85,B 0,C 180,E1 -5973.994,E2 -5973.994} C_VEL
LIN {X 0,Y 502.78,Z 411.482,A -85,B 0,C 180,E1 -5977.178,E2 -5977.178} C_VEL
LIN {X 0,Y 502.79,Z 411.48,A -85,B 0,C 180,E1 -5980.015,E2 -5980.015} C_VEL
LIN {X 0,Y 502.805,Z 411.483,A -85,B 0,C 180,E1 -5982.199,E2 -5982.199} C_VEL
LIN {X 0,Y 502.803,Z 411.482,A -85,B 0,C 180,E1 -5985.468,E2 -5985.468} C_VEL
LIN {X 0,Y 502.822,Z 411.482,A -85,B 0,C 180,E1 -5988.934,E2 -5988.934} C_VEL
LIN {X 0,Y 502.85,Z 411.486,A -85,B 0,C 180,E1 -5989.86,E2 -5989.86} C_VEL
LIN {X 0,Y 503.903,Z 418.168,A -85,B 0,C 180,E1 -5991.767,E2 -5991.767} C_VEL
LIN {X 0,Y 503.774,Z 426.523,A -85,B 0,C 180,E1 -5994.131,E2 -5994.131} C_VEL
LIN {X 0,Y 503.655,Z 431.581,A -85,B 0,C 180,E1 -5995.59,E2 -5995.59} C_VEL
LIN {X 0,Y 502.951,Z 433.83,A -85,B 0,C 180,E1 -5996.207,E2 -5996.207} C_VEL
LIN {X 0,Y 497.205,Z 441.646,A -85,B 0,C 180,E1 -5998.195,E2 -5998.195} C_VEL
LIN {X 0,Y 496.553,Z 443.88,A -85,B 0,C 180,E1 -5998.824,E2 -5998.824} C_VEL
LIN {X 0,Y 496.422,Z 453.804,A -85,B 0,C 180,E1 -6001.763,E2 -6001.763} C_VEL
LIN {X 0,Y 496.134,Z 464.367,A -85,B 0,C 180,E1 -6004.851,E2 -6004.851} C_VEL
LIN {X 0,Y 495.972,Z 475.199,A -85,B 0,C 180,E1 -6007.944,E2 -6007.944} C_VEL
LIN {X 0,Y 495.801,Z 486.063,A -85,B 0,C 180,E1 -6010.972,E2 -6010.972} C_VEL
LIN {X 0,Y 495.714,Z 491.516,A -85,B 0,C 180,E1 -6012.493,E2 -6012.493} C_VEL
LIN {X 0,Y 499.115,Z 508.228,A -85,B 0,C 180,E1 -6012.972,E2 -6012.972} C_VEL
LIN {X 0,Y 498.776,Z 521.699,A -85,B 0,C 180,E1 -6013.415,E2 -6013.415} C_VEL
LIN {X 0,Y 498.374,Z 535.398,A -85,B 0,C 180,E1 -6014.039,E2 -6014.039} C_VEL
LIN {X 0,Y 497.898,Z 547.68,A -85,B 0,C 180,E1 -6014.758,E2 -6014.758} C_VEL
LIN {X 0,Y 497.379,Z 559.031,A -85,B 0,C 180,E1 -6015.579,E2 -6015.579} C_VEL
LIN {X 0,Y 496.839,Z 570.638,A -85,B 0,C 180,E1 -6016.607,E2 -6016.607} C_VEL
LIN {X 0,Y 496.346,Z 581.15,A -85,B 0,C 180,E1 -6017.737,E2 -6017.737} C_VEL
LIN {X 0,Y 496.039,Z 590.638,A -85,B 0,C 180,E1 -6018.973,E2 -6018.973} C_VEL
LIN {X 0,Y 495.674,Z 598.511,A -85,B 0,C 180,E1 -6020.204,E2 -6020.204} C_VEL
LIN {X 0,Y 495.42,Z 605.065,A -85,B 0,C 180,E1 -6021.434,E2 -6021.434} C_VEL
LIN {X 0,Y 495.181,Z 610.506,A -85,B 0,C 180,E1 -6022.661,E2 -6022.661} C_VEL
LIN {X 0,Y 495.151,Z 616.204,A -85,B 0,C 180,E1 -6024.298,E2 -6024.298} C_VEL
LIN {X 0,Y 495.017,Z 620.352,A -85,B 0,C 180,E1 -6025.929,E2 -6025.929} C_VEL
LIN {X 0,Y 494.973,Z 623.069,A -85,B 0,C 180,E1 -6027.559,E2 -6027.559} C_VEL
LIN {X 0,Y 494.908,Z 624.436,A -85,B 0,C 180,E1 -6029.186,E2 -6029.186} C_VEL
LIN {X 0,Y 494.908,Z 624.48,A -85,B 0,C 180,E1 -6030.814,E2 -6030.814} C_VEL
LIN {X 0,Y 494.972,Z 623.189,A -85,B 0,C 180,E1 -6032.441,E2 -6032.441} C_VEL
LIN {X 0,Y 495.016,Z 620.542,A -85,B 0,C 180,E1 -6034.071,E2 -6034.071} C_VEL
LIN {X 0,Y 495.148,Z 616.473,A -85,B 0,C 180,E1 -6035.702,E2 -6035.702} C_VEL
LIN {X 0,Y 495.18,Z 610.856,A -85,B 0,C 180,E1 -6037.339,E2 -6037.339} C_VEL
LIN {X 0,Y 495.394,Z 605.498,A -85,B 0,C 180,E1 -6038.567,E2 -6038.567} C_VEL
LIN {X 0,Y 495.661,Z 597.829,A -85,B 0,C 180,E1 -6040.003,E2 -6040.003} C_VEL
LIN {X 0,Y 496.044,Z 589.815,A -85,B 0,C 180,E1 -6041.234,E2 -6041.234} C_VEL
LIN {X 0,Y 496.464,Z 580.337,A -85,B 0,C 180,E1 -6042.446,E2 -6042.446} C_VEL
LIN {X 0,Y 496.937,Z 569.452,A -85,B 0,C 180,E1 -6043.599,E2 -6043.599} C_VEL
LIN {X 0,Y 497.445,Z 557.583,A -85,B 0,C 180,E1 -6044.628,E2 -6044.628} C_VEL
LIN {X 0,Y 497.963,Z 545.9,A -85,B 0,C 180,E1 -6045.45,E2 -6045.45} C_VEL
LIN {X 0,Y 498.475,Z 532.029,A -85,B 0,C 180,E1 -6046.221,E2 -6046.221} C_VEL
LIN {X 0,Y 498.923,Z 517.691,A -85,B 0,C 180,E1 -6046.819,E2 -6046.819} C_VEL
LIN {X 0,Y 498.963,Z 507.73,A -85,B 0,C 180,E1 -6047.136,E2 -6047.136} C_VEL
LIN {X 0,Y 496.005,Z 493.225,A -85,B 0,C 180,E1 -6047.552,E2 -6047.552} C_VEL
LIN {X 0,Y 495.69,Z 491.512,A -85,B 0,C 180,E1 -6047.602,E2 -6047.602} C_VEL
LIN {X 0,Y 495.866,Z 481.833,A -85,B 0,C 180,E1 -6050.294,E2 -6050.294} C_VEL
LIN {X 0,Y 495.998,Z 472.418,A -85,B 0,C 180,E1 -6052.925,E2 -6052.925} C_VEL
LIN {X 0,Y 496.208,Z 461.589,A -85,B 0,C 180,E1 -6056.044,E2 -6056.044} C_VEL
LIN {X 0,Y 496.408,Z 452.315,A -85,B 0,C 180,E1 -6058.774,E2 -6058.774} C_VEL
LIN {X 0,Y 496.558,Z 442.842,A -85,B 0,C 180,E1 -6061.579,E2 -6061.579} C_VEL
LIN {X 0,Y 496.693,Z 431.74,A -85,B 0,C 180,E1 -6064.847,E2 -6064.847} C_VEL
LIN {X 0,Y 496.99,Z 422.057,A -85,B 0,C 180,E1 -6067.636,E2 -6067.636} C_VEL
LIN {X 0,Y 496.718,Z 417.659,A -85,B 0,C 180,E1 -6068.905,E2 -6068.905} C_VEL
LIN {X 0,Y 495.79,Z 412.357,A -85,B 0,C 180,E1 -6070.437,E2 -6070.437} C_VEL
LIN {X 0,Y 495.731,Z 412.362,A -85,B 0,C 180,E1 -6073.695,E2 -6073.695} C_VEL
LIN {X 0,Y 495.737,Z 412.36,A -85,B 0,C 180,E1 -6076.305,E2 -6076.305} C_VEL
LIN {X 0,Y 495.769,Z 412.361,A -85,B 0,C 180,E1 -6079.3,E2 -6079.3} C_VEL
LIN {X 0,Y 495.733,Z 412.361,A -85,B 0,C 180,E1 -6082.438,E2 -6082.438} C_VEL
LIN {X 0,Y 495.786,Z 412.353,A -85,B 0,C 180,E1 -6085.457,E2 -6085.457} C_VEL
LIN {X 0,Y 495.758,Z 412.357,A -85,B 0,C 180,E1 -6088.364,E2 -6088.364} C_VEL
LIN {X 0,Y 495.791,Z 412.356,A -85,B 0,C 180,E1 -6091.506,E2 -6091.506} C_VEL
LIN {X 0,Y 495.793,Z 412.355,A -85,B 0,C 180,E1 -6093.932,E2 -6093.932} C_VEL
LIN {X 0,Y 495.761,Z 412.356,A -85,B 0,C 180,E1 -6097.14,E2 -6097.14} C_VEL
LIN {X 0,Y 495.812,Z 412.395,A -85,B 0,C 180,E1 -6100.478,E2 -6100.478} C_VEL
LIN {X 0,Y 499.681,Z 424.675,A -85,B 0,C 180,E1 -6101.125,E2 -6101.125} C_VEL
LIN {X 0,Y 499.24,Z 439.411,A -85,B 0,C 180,E1 -6101.874,E2 -6101.874} C_VEL
LIN {X 0,Y 498.686,Z 452.153,A -85,B 0,C 180,E1 -6102.679,E2 -6102.679} C_VEL
LIN {X 0,Y 497.988,Z 465.759,A -85,B 0,C 180,E1 -6103.733,E2 -6103.733} C_VEL
LIN {X 0,Y 497.427,Z 477.616,A -85,B 0,C 180,E1 -6104.848,E2 -6104.848} C_VEL
LIN {X 0,Y 496.924,Z 488.607,A -85,B 0,C 180,E1 -6106.088,E2 -6106.088} C_VEL
LIN {X 0,Y 496.399,Z 497.869,A -85,B 0,C 180,E1 -6107.323,E2 -6107.323} C_VEL
LIN {X 0,Y 496.063,Z 506.903,A -85,B 0,C 180,E1 -6108.767,E2 -6108.767} C_VEL
LIN {X 0,Y 495.663,Z 514.422,A -85,B 0,C 180,E1 -6110.203,E2 -6110.203} C_VEL
LIN {X 0,Y 495.448,Z 521.393,A -85,B 0,C 180,E1 -6111.845,E2 -6111.845} C_VEL
LIN {X 0,Y 495.251,Z 526.827,A -85,B 0,C 180,E1 -6113.481,E2 -6113.481} C_VEL
LIN {X 0,Y 495.119,Z 530.969,A -85,B 0,C 180,E1 -6115.114,E2 -6115.114} C_VEL
LIN {X 0,Y 495.095,Z 533.882,A -85,B 0,C 180,E1 -6116.745,E2 -6116.745} C_VEL
LIN {X 0,Y 494.995,Z 535.62,A -85,B 0,C 180,E1 -6118.373,E2 -6118.373} C_VEL
LIN {X 0,Y 494.951,Z 536.228,A -85,B 0,C 180,E1 -6120,E2 -6120} C_VEL
LIN {X 0,Y 495.005,Z 535.719,A -85,B 0,C 180,E1 -6121.627,E2 -6121.627} C_VEL
LIN {X 0,Y 495.095,Z 534.107,A -85,B 0,C 180,E1 -6123.255,E2 -6123.255} C_VEL
LIN {X 0,Y 495.121,Z 531.356,A -85,B 0,C 180,E1 -6124.886,E2 -6124.886} C_VEL
LIN {X 0,Y 495.345,Z 526.807,A -85,B 0,C 180,E1 -6126.701,E2 -6126.701} C_VEL
LIN {X 0,Y 495.481,Z 522.024,A -85,B 0,C 180,E1 -6128.154,E2 -6128.154} C_VEL
LIN {X 0,Y 495.716,Z 515.225,A -85,B 0,C 180,E1 -6129.795,E2 -6129.795} C_VEL
LIN {X 0,Y 496.123,Z 506.663,A -85,B 0,C 180,E1 -6131.439,E2 -6131.439} C_VEL
LIN {X 0,Y 496.501,Z 497.502,A -85,B 0,C 180,E1 -6132.882,E2 -6132.882} C_VEL
LIN {X 0,Y 496.983,Z 488.091,A -85,B 0,C 180,E1 -6134.119,E2 -6134.119} C_VEL
LIN {X 0,Y 497.515,Z 476.824,A -85,B 0,C 180,E1 -6135.359,E2 -6135.359} C_VEL
LIN {X 0,Y 498.093,Z 465.594,A -85,B 0,C 180,E1 -6136.391,E2 -6136.391} C_VEL
LIN {X 0,Y 498.597,Z 453.436,A -85,B 0,C 180,E1 -6137.324,E2 -6137.324} C_VEL
LIN {X 0,Y 499.174,Z 438.977,A -85,B 0,C 180,E1 -6138.219,E2 -6138.219} C_VEL
LIN {X 0,Y 499.576,Z 425.592,A -85,B 0,C 180,E1 -6138.878,E2 -6138.878} C_VEL
LIN {X 0,Y 498.701,Z 421.775,A -85,B 0,C 180,E1 -6139.07,E2 -6139.07} C_VEL
LIN {X 0,Y 495.792,Z 412.354,A -85,B 0,C 180,E1 -6139.563,E2 -6139.563} C_VEL
LIN {X 0,Y 495.761,Z 412.354,A -85,B 0,C 180,E1 -6142.861,E2 -6142.861} C_VEL
LIN {X 0,Y 495.783,Z 412.359,A -85,B 0,C 180,E1 -6146.068,E2 -6146.068} C_VEL
LIN {X 0,Y 495.774,Z 412.353,A -85,B 0,C 180,E1 -6148.815,E2 -6148.815} C_VEL
LIN {X 0,Y 495.761,Z 412.359,A -85,B 0,C 180,E1 -6151.726,E2 -6151.726} C_VEL
LIN {X 0,Y 495.77,Z 412.352,A -85,B 0,C 180,E1 -6154.694,E2 -6154.694} C_VEL
LIN {X 0,Y 495.731,Z 412.363,A -85,B 0,C 180,E1 -6157.562,E2 -6157.562} C_VEL
LIN {X 0,Y 495.768,Z 412.354,A -85,B 0,C 180,E1 -6160.7,E2 -6160.7} C_VEL
LIN {X 0,Y 495.786,Z 412.356,A -85,B 0,C 180,E1 -6163.995,E2 -6163.995} C_VEL
LIN {X 0,Y 495.819,Z 412.463,A -85,B 0,C 180,E1 -6164.345,E2 -6164.345} C_VEL
LIN {X 0,Y 495.875,Z 415.937,A -85,B 0,C 180,E1 -6165.56,E2 -6165.56} C_VEL
LIN {X 0,Y 495.692,Z 428.689,A -85,B 0,C 180,E1 -6169.66,E2 -6169.66} C_VEL
LIN {X 0,Y 495.915,Z 438.06,A -85,B 0,C 180,E1 -6172.525,E2 -6172.525} C_VEL
LIN {X 0,Y 496.092,Z 447.945,A -85,B 0,C 180,E1 -6175.482,E2 -6175.482} C_VEL
LIN {X 0,Y 496.119,Z 457.771,A -85,B 0,C 180,E1 -6178.39,E2 -6178.39} C_VEL
LIN {X 0,Y 496.17,Z 468.094,A -85,B 0,C 180,E1 -6181.426,E2 -6181.426} C_VEL
LIN {X 0,Y 496,Z 478.068,A -85,B 0,C 180,E1 -6184.395,E2 -6184.395} C_VEL
LIN {X 0,Y 495.871,Z 487.12,A -85,B 0,C 180,E1 -6187.109,E2 -6187.109} C_VEL
LIN {X 0,Y 495.707,Z 494.681,A -85,B 0,C 180,E1 -6189.723,E2 -6189.723} C_VEL
LIN {X 0,Y 495.56,Z 502.636,A -85,B 0,C 180,E1 -6192.461,E2 -6192.461} C_VEL
LIN {X 0,Y 498.687,Z 517.559,A -85,B 0,C 180,E1 -6192.894,E2 -6192.894} C_VEL
LIN {X 0,Y 499.091,Z 520.793,A -85,B 0,C 180,E1 -6192.999,E2 -6192.999} C_VEL
LIN {X 0,Y 498.765,Z 533.411,A -85,B 0,C 180,E1 -6193.441,E2 -6193.441} C_VEL
LIN {X 0,Y 498.285,Z 546.185,A -85,B 0,C 180,E1 -6194.036,E2 -6194.036} C_VEL
LIN {X 0,Y 497.804,Z 559.75,A -85,B 0,C 180,E1 -6194.86,E2 -6194.86} C_VEL
LIN {X 0,Y 497.221,Z 571.927,A -85,B 0,C 180,E1 -6195.783,E2 -6195.783} C_VEL
LIN {X 0,Y 496.733,Z 582.997,A -85,B 0,C 180,E1 -6196.812,E2 -6196.812} C_VEL
LIN {X 0,Y 496.303,Z 593.133,A -85,B 0,C 180,E1 -6197.95,E2 -6197.95} C_VEL
LIN {X 0,Y 495.919,Z 602.224,A -85,B 0,C 180,E1 -6199.177,E2 -6199.177} C_VEL
LIN {X 0,Y 495.548,Z 610.943,A -85,B 0,C 180,E1 -6200.613,E2 -6200.613} C_VEL
LIN {X 0,Y 495.336,Z 617.074,A -85,B 0,C 180,E1 -6201.843,E2 -6201.843} C_VEL
LIN {X 0,Y 495.171,Z 622.116,A -85,B 0,C 180,E1 -6203.071,E2 -6203.071} C_VEL
LIN {X 0,Y 495.105,Z 627.397,A -85,B 0,C 180,E1 -6204.706,E2 -6204.706} C_VEL
LIN {X 0,Y 495.013,Z 630.312,A -85,B 0,C 180,E1 -6205.929,E2 -6205.929} C_VEL
LIN {X 0,Y 494.972,Z 632.996,A -85,B 0,C 180,E1 -6207.559,E2 -6207.559} C_VEL
LIN {X 0,Y 494.908,Z 634.332,A -85,B 0,C 180,E1 -6209.186,E2 -6209.186} C_VEL
LIN {X 0,Y 494.908,Z 634.33,A -85,B 0,C 180,E1 -6210.814,E2 -6210.814} C_VEL
LIN {X 0,Y 494.972,Z 632.995,A -85,B 0,C 180,E1 -6212.441,E2 -6212.441} C_VEL
LIN {X 0,Y 495.013,Z 630.314,A -85,B 0,C 180,E1 -6214.071,E2 -6214.071} C_VEL
LIN {X 0,Y 495.129,Z 626.216,A -85,B 0,C 180,E1 -6215.702,E2 -6215.702} C_VEL
LIN {X 0,Y 495.18,Z 620.553,A -85,B 0,C 180,E1 -6217.339,E2 -6217.339} C_VEL
LIN {X 0,Y 495.428,Z 614.141,A -85,B 0,C 180,E1 -6218.772,E2 -6218.772} C_VEL
LIN {X 0,Y 495.711,Z 606.166,A -85,B 0,C 180,E1 -6220.208,E2 -6220.208} C_VEL
LIN {X 0,Y 496.127,Z 597.85,A -85,B 0,C 180,E1 -6221.439,E2 -6221.439} C_VEL
LIN {X 0,Y 496.506,Z 588.191,A -85,B 0,C 180,E1 -6222.632,E2 -6222.632} C_VEL
LIN {X 0,Y 497.031,Z 576.62,A -85,B 0,C 180,E1 -6223.805,E2 -6223.805} C_VEL
LIN {X 0,Y 497.487,Z 565.481,A -85,B 0,C 180,E1 -6224.731,E2 -6224.731} C_VEL
LIN {X 0,Y 498.039,Z 553.366,A -85,B 0,C 180,E1 -6225.552,E2 -6225.552} C_VEL
LIN {X 0,Y 498.547,Z 539.989,A -85,B 0,C 180,E1 -6226.271,E2 -6226.271} C_VEL
LIN {X 0,Y 498.919,Z 526.077,A -85,B 0,C 180,E1 -6226.834,E2 -6226.834} C_VEL
LIN {X 0,Y 498.905,Z 518.765,A -85,B 0,C 180,E1 -6227.065,E2 -6227.065} C_VEL
LIN {X 0,Y 495.834,Z 504.125,A -85,B 0,C 180,E1 -6227.503,E2 -6227.503} C_VEL
LIN {X 0,Y 495.554,Z 502.439,A -85,B 0,C 180,E1 -6227.56,E2 -6227.56} C_VEL
LIN {X 0,Y 495.74,Z 493.319,A -85,B 0,C 180,E1 -6230.758,E2 -6230.758} C_VEL
LIN {X 0,Y 495.907,Z 485.699,A -85,B 0,C 180,E1 -6233.379,E2 -6233.379} C_VEL
LIN {X 0,Y 496.081,Z 476.569,A -85,B 0,C 180,E1 -6236.431,E2 -6236.431} C_VEL
LIN {X 0,Y 496.331,Z 468.408,A -85,B 0,C 180,E1 -6239.243,E2 -6239.243} C_VEL
LIN {X 0,Y 496.478,Z 459.144,A -85,B 0,C 180,E1 -6242.542,E2 -6242.542} C_VEL
LIN {X 0,Y 496.675,Z 450.111,A -85,B 0,C 180,E1 -6245.855,E2 -6245.855} C_VEL
LIN {X 0,Y 496.822,Z 442.089,A -85,B 0,C 180,E1 -6248.92,E2 -6248.92} C_VEL
LIN {X 0,Y 497.024,Z 435.188,A -85,B 0,C 180,E1 -6251.651,E2 -6251.651} C_VEL
LIN {X 0,Y 497.351,Z 426.925,A -85,B 0,C 180,E1 -6255.046,E2 -6255.046} C_VEL
LIN {X 0,Y 497.299,Z 421.692,A -85,B 0,C 180,E1 -6257.297,E2 -6257.297} C_VEL
LIN {X 0,Y 496.422,Z 416.102,A -85,B 0,C 180,E1 -6259.862,E2 -6259.862} C_VEL
LIN {X 0,Y 495.77,Z 412.356,A -85,B 0,C 180,E1 -6261.67,E2 -6261.67} C_VEL
LIN {X 0,Y 495.757,Z 412.356,A -85,B 0,C 180,E1 -6264.463,E2 -6264.463} C_VEL
LIN {X 0,Y 495.769,Z 412.356,A -85,B 0,C 180,E1 -6267.406,E2 -6267.406} C_VEL
LIN {X 0,Y 495.768,Z 412.357,A -85,B 0,C 180,E1 -6270.254,E2 -6270.254} C_VEL
LIN {X 0,Y 495.825,Z 412.343,A -85,B 0,C 180,E1 -6273.251,E2 -6273.251} C_VEL
LIN {X 0,Y 495.755,Z 412.357,A -85,B 0,C 180,E1 -6275.725,E2 -6275.725} C_VEL
LIN {X 0,Y 495.75,Z 412.354,A -85,B 0,C 180,E1 -6278.371,E2 -6278.371} C_VEL
LIN {X 0,Y 495.787,Z 412.351,A -85,B 0,C 180,E1 -6280.972,E2 -6280.972} C_VEL
LIN {X 0,Y 495.783,Z 412.353,A -85,B 0,C 180,E1 -6283.53,E2 -6283.53} C_VEL
LIN {X 0,Y 495.796,Z 412.346,A -85,B 0,C 180,E1 -6286.056,E2 -6286.056} C_VEL
LIN {X 0,Y 495.854,Z 412.343,A -85,B 0,C 180,E1 -6288.555,E2 -6288.555} C_VEL
LIN {X 0,Y 495.839,Z 412.34,A -85,B 0,C 180,E1 -6291.852,E2 -6291.852} C_VEL
LIN {X 0,Y 495.899,Z 412.339,A -85,B 0,C 180,E1 -6294.307,E2 -6294.307} C_VEL
LIN {X 0,Y 495.995,Z 412.321,A -85,B 0,C 180,E1 -6297.564,E2 -6297.564} C_VEL
LIN {X 0,Y 496.001,Z 412.33,A -85,B 0,C 180,E1 -6300,E2 -6300} C_VEL
LIN {X 0,Y 495.995,Z 412.322,A -85,B 0,C 180,E1 -6302.436,E2 -6302.436} C_VEL
LIN {X 0,Y 495.898,Z 412.34,A -85,B 0,C 180,E1 -6305.694,E2 -6305.694} C_VEL
LIN {X 0,Y 495.876,Z 412.335,A -85,B 0,C 180,E1 -6308.148,E2 -6308.148} C_VEL
LIN {X 0,Y 495.854,Z 412.344,A -85,B 0,C 180,E1 -6311.445,E2 -6311.445} C_VEL
LIN {X 0,Y 495.792,Z 412.349,A -85,B 0,C 180,E1 -6314.783,E2 -6314.783} C_VEL
LIN {X 0,Y 495.789,Z 412.351,A -85,B 0,C 180,E1 -6317.319,E2 -6317.319} C_VEL
LIN {X 0,Y 495.781,Z 412.355,A -85,B 0,C 180,E1 -6319.89,E2 -6319.89} C_VEL
LIN {X 0,Y 495.761,Z 412.354,A -85,B 0,C 180,E1 -6322.861,E2 -6322.861} C_VEL
LIN {X 0,Y 495.783,Z 412.351,A -85,B 0,C 180,E1 -6326.068,E2 -6326.068} C_VEL
LIN {X 0,Y 495.774,Z 412.355,A -85,B 0,C 180,E1 -6328.815,E2 -6328.815} C_VEL
LIN {X 0,Y 495.758,Z 412.359,A -85,B 0,C 180,E1 -6331.725,E2 -6331.725} C_VEL
LIN {X 0,Y 495.771,Z 412.357,A -85,B 0,C 180,E1 -6334.694,E2 -6334.694} C_VEL
LIN {X 0,Y 495.731,Z 412.362,A -85,B 0,C 180,E1 -6337.562,E2 -6337.562} C_VEL
LIN {X 0,Y 495.769,Z 412.359,A -85,B 0,C 180,E1 -6340.7,E2 -6340.7} C_VEL
LIN {X 0,Y 495.737,Z 412.363,A -85,B 0,C 180,E1 -6343.696,E2 -6343.696} C_VEL
LIN {X 0,Y 495.731,Z 412.363,A -85,B 0,C 180,E1 -6346.305,E2 -6346.305} C_VEL
LIN {X 0,Y 495.827,Z 412.412,A -85,B 0,C 180,E1 -6349.672,E2 -6349.672} C_VEL
LIN {X 0,Y 496.882,Z 418.762,A -85,B 0,C 180,E1 -6351.512,E2 -6351.512} C_VEL
LIN {X 0,Y 496.891,Z 425.905,A -85,B 0,C 180,E1 -6353.555,E2 -6353.555} C_VEL
LIN {X 0,Y 496.614,Z 437.842,A -85,B 0,C 180,E1 -6357.04,E2 -6357.04} C_VEL
LIN {X 0,Y 496.553,Z 443.88,A -85,B 0,C 180,E1 -6358.824,E2 -6358.824} C_VEL
LIN {X 0,Y 495.899,Z 446.11,A -85,B 0,C 180,E1 -6359.45,E2 -6359.45} C_VEL
LIN {X 0,Y 493.028,Z 449.98,A -85,B 0,C 180,E1 -6360.454,E2 -6360.454} C_VEL
LIN {X 0,Y 490.098,Z 453.858,A -85,B 0,C 180,E1 -6361.468,E2 -6361.468} C_VEL
LIN {X 0,Y 489.375,Z 456.104,A -85,B 0,C 180,E1 -6362.106,E2 -6362.106} C_VEL
LIN {X 0,Y 489.063,Z 467.192,A -85,B 0,C 180,E1 -6365.371,E2 -6365.371} C_VEL
LIN {X 0,Y 488.911,Z 476.492,A -85,B 0,C 180,E1 -6368.053,E2 -6368.053} C_VEL
LIN {X 0,Y 488.737,Z 487.445,A -85,B 0,C 180,E1 -6371.122,E2 -6371.122} C_VEL
LIN {X 0,Y 488.656,Z 491.5,A -85,B 0,C 180,E1 -6372.24,E2 -6372.24} C_VEL
LIN {X 0,Y 491.856,Z 507.045,A -85,B 0,C 180,E1 -6372.682,E2 -6372.682} C_VEL
LIN {X 0,Y 492.309,Z 510.241,A -85,B 0,C 180,E1 -6372.79,E2 -6372.79} C_VEL
LIN {X 0,Y 491.895,Z 523.919,A -85,B 0,C 180,E1 -6373.27,E2 -6373.27} C_VEL
LIN {X 0,Y 491.49,Z 537.353,A -85,B 0,C 180,E1 -6373.916,E2 -6373.916} C_VEL
LIN {X 0,Y 490.912,Z 550.792,A -85,B 0,C 180,E1 -6374.748,E2 -6374.748} C_VEL
LIN {X 0,Y 490.406,Z 561.594,A -85,B 0,C 180,E1 -6375.582,E2 -6375.582} C_VEL
LIN {X 0,Y 489.841,Z 572.779,A -85,B 0,C 180,E1 -6376.623,E2 -6376.623} C_VEL
LIN {X 0,Y 489.29,Z 583.007,A -85,B 0,C 180,E1 -6377.775,E2 -6377.775} C_VEL
LIN {X 0,Y 488.962,Z 592.143,A -85,B 0,C 180,E1 -6379.021,E2 -6379.021} C_VEL
LIN {X 0,Y 488.604,Z 599.776,A -85,B 0,C 180,E1 -6380.27,E2 -6380.27} C_VEL
LIN {X 0,Y 488.281,Z 607.081,A -85,B 0,C 180,E1 -6381.724,E2 -6381.724} C_VEL
LIN {X 0,Y 488.096,Z 613.616,A -85,B 0,C 180,E1 -6383.385,E2 -6383.385} C_VEL
LIN {X 0,Y 488.046,Z 617.471,A -85,B 0,C 180,E1 -6384.629,E2 -6384.629} C_VEL
LIN {X 0,Y 487.918,Z 620.411,A -85,B 0,C 180,E1 -6385.87,E2 -6385.87} C_VEL
LIN {X 0,Y 487.886,Z 623.128,A -85,B 0,C 180,E1 -6387.523,E2 -6387.523} C_VEL
LIN {X 0,Y 487.831,Z 624.495,A -85,B 0,C 180,E1 -6389.175,E2 -6389.175} C_VEL
LIN {X 0,Y 487.831,Z 624.538,A -85,B 0,C 180,E1 -6390.825,E2 -6390.825} C_VEL
LIN {X 0,Y 487.885,Z 623.246,A -85,B 0,C 180,E1 -6392.477,E2 -6392.477} C_VEL
LIN {X 0,Y 487.918,Z 620.598,A -85,B 0,C 180,E1 -6394.13,E2 -6394.13} C_VEL
LIN {X 0,Y 488.064,Z 616.527,A -85,B 0,C 180,E1 -6395.785,E2 -6395.785} C_VEL
LIN {X 0,Y 488.132,Z 610.909,A -85,B 0,C 180,E1 -6397.445,E2 -6397.445} C_VEL
LIN {X 0,Y 488.361,Z 605.549,A -85,B 0,C 180,E1 -6398.691,E2 -6398.691} C_VEL
LIN {X 0,Y 488.616,Z 597.878,A -85,B 0,C 180,E1 -6400.148,E2 -6400.148} C_VEL
LIN {X 0,Y 489.061,Z 589.86,A -85,B 0,C 180,E1 -6401.396,E2 -6401.396} C_VEL
LIN {X 0,Y 489.495,Z 580.204,A -85,B 0,C 180,E1 -6402.648,E2 -6402.648} C_VEL
LIN {X 0,Y 489.998,Z 569.491,A -85,B 0,C 180,E1 -6403.795,E2 -6403.795} C_VEL
LIN {X 0,Y 490.536,Z 557.615,A -85,B 0,C 180,E1 -6404.839,E2 -6404.839} C_VEL
LIN {X 0,Y 491.09,Z 545.925,A -85,B 0,C 180,E1 -6405.671,E2 -6405.671} C_VEL
LIN {X 0,Y 491.656,Z 532.042,A -85,B 0,C 180,E1 -6406.452,E2 -6406.452} C_VEL
LIN {X 0,Y 492.123,Z 517.862,A -85,B 0,C 180,E1 -6407.052,E2 -6407.052} C_VEL
LIN {X 0,Y 492.209,Z 509.026,A -85,B 0,C 180,E1 -6407.342,E2 -6407.342} C_VEL
LIN {X 0,Y 489.202,Z 494.094,A -85,B 0,C 180,E1 -6407.789,E2 -6407.789} C_VEL
LIN {X 0,Y 488.647,Z 491.374,A -85,B 0,C 180,E1 -6407.878,E2 -6407.878} C_VEL
LIN {X 0,Y 488.828,Z 480.695,A -85,B 0,C 180,E1 -6410.849,E2 -6410.849} C_VEL
LIN {X 0,Y 488.974,Z 470.594,A -85,B 0,C 180,E1 -6413.731,E2 -6413.731} C_VEL
LIN {X 0,Y 489.258,Z 460.269,A -85,B 0,C 180,E1 -6416.749,E2 -6416.749} C_VEL
LIN {X 0,Y 489.443,Z 450.383,A -85,B 0,C 180,E1 -6419.696,E2 -6419.696} C_VEL
LIN {X 0,Y 489.629,Z 440.781,A -85,B 0,C 180,E1 -6422.565,E2 -6422.565} C_VEL
LIN {X 0,Y 489.821,Z 429.065,A -85,B 0,C 180,E1 -6426.035,E2 -6426.035} C_VEL
LIN {X 0,Y 490.01,Z 422,A -85,B 0,C 180,E1 -6428.078,E2 -6428.078} C_VEL
LIN {X 0,Y 489.281,Z 416.373,A -85,B 0,C 180,E1 -6429.731,E2 -6429.731} C_VEL
LIN {X 0,Y 488.754,Z 413.233,A -85,B 0,C 180,E1 -6430.659,E2 -6430.659} C_VEL
LIN {X 0,Y 488.702,Z 413.237,A -85,B 0,C 180,E1 -6434.024,E2 -6434.024} C_VEL
LIN {X 0,Y 488.734,Z 413.238,A -85,B 0,C 180,E1 -6437.171,E2 -6437.171} C_VEL
LIN {X 0,Y 488.735,Z 413.236,A -85,B 0,C 180,E1 -6439.677,E2 -6439.677} C_VEL
LIN {X 0,Y 488.684,Z 413.239,A -85,B 0,C 180,E1 -6442.841,E2 -6442.841} C_VEL
LIN {X 0,Y 488.736,Z 413.228,A -85,B 0,C 180,E1 -6445.887,E2 -6445.887} C_VEL
LIN {X 0,Y 488.697,Z 413.237,A -85,B 0,C 180,E1 -6448.82,E2 -6448.82} C_VEL
LIN {X 0,Y 488.748,Z 413.232,A -85,B 0,C 180,E1 -6451.671,E2 -6451.671} C_VEL
LIN {X 0,Y 488.75,Z 413.23,A -85,B 0,C 180,E1 -6454.444,E2 -6454.444} C_VEL
LIN {X 0,Y 488.724,Z 413.233,A -85,B 0,C 180,E1 -6457.153,E2 -6457.153} C_VEL
LIN {X 0,Y 488.75,Z 413.248,A -85,B 0,C 180,E1 -6460.223,E2 -6460.223} C_VEL
LIN {X 0,Y 492.928,Z 426.521,A -85,B 0,C 180,E1 -6460.946,E2 -6460.946} C_VEL
LIN {X 0,Y 492.417,Z 440.941,A -85,B 0,C 180,E1 -6461.7,E2 -6461.7} C_VEL
LIN {X 0,Y 491.793,Z 453.834,A -85,B 0,C 180,E1 -6462.536,E2 -6462.536} C_VEL
LIN {X 0,Y 491.135,Z 466.823,A -85,B 0,C 180,E1 -6463.567,E2 -6463.567} C_VEL
LIN {X 0,Y 490.569,Z 478.011,A -85,B 0,C 180,E1 -6464.631,E2 -6464.631} C_VEL
LIN {X 0,Y 490.028,Z 489.081,A -85,B 0,C 180,E1 -6465.888,E2 -6465.888} C_VEL
LIN {X 0,Y 489.395,Z 499.79,A -85,B 0,C 180,E1 -6467.35,E2 -6467.35} C_VEL
LIN {X 0,Y 489.064,Z 508.656,A -85,B 0,C 180,E1 -6468.814,E2 -6468.814} C_VEL
LIN {X 0,Y 488.576,Z 516.923,A -85,B 0,C 180,E1 -6470.478,E2 -6470.478} C_VEL
LIN {X 0,Y 488.376,Z 523.527,A -85,B 0,C 180,E1 -6472.142,E2 -6472.142} C_VEL
LIN {X 0,Y 488.189,Z 528.346,A -85,B 0,C 180,E1 -6473.675,E2 -6473.675} C_VEL
LIN {X 0,Y 488.096,Z 531.669,A -85,B 0,C 180,E1 -6475.044,E2 -6475.044} C_VEL
LIN {X 0,Y 488.051,Z 534.603,A -85,B 0,C 180,E1 -6476.698,E2 -6476.698} C_VEL
LIN {X 0,Y 487.939,Z 536.371,A -85,B 0,C 180,E1 -6478.349,E2 -6478.349} C_VEL
LIN {X 0,Y 487.895,Z 537.009,A -85,B 0,C 180,E1 -6480,E2 -6480} C_VEL
LIN {X 0,Y 487.952,Z 536.506,A -85,B 0,C 180,E1 -6481.651,E2 -6481.651} C_VEL
LIN {X 0,Y 488.052,Z 534.879,A -85,B 0,C 180,E1 -6483.302,E2 -6483.302} C_VEL
LIN {X 0,Y 488.1,Z 532.116,A -85,B 0,C 180,E1 -6484.956,E2 -6484.956} C_VEL
LIN {X 0,Y 488.324,Z 527.688,A -85,B 0,C 180,E1 -6486.756,E2 -6486.756} C_VEL
LIN {X 0,Y 488.498,Z 522.766,A -85,B 0,C 180,E1 -6488.272,E2 -6488.272} C_VEL
LIN {X 0,Y 488.729,Z 515.922,A -85,B 0,C 180,E1 -6489.937,E2 -6489.937} C_VEL
LIN {X 0,Y 489.144,Z 508.528,A -85,B 0,C 180,E1 -6491.394,E2 -6491.394} C_VEL
LIN {X 0,Y 489.54,Z 499.563,A -85,B 0,C 180,E1 -6492.857,E2 -6492.857} C_VEL
LIN {X 0,Y 490.043,Z 490.356,A -85,B 0,C 180,E1 -6494.111,E2 -6494.111} C_VEL
LIN {X 0,Y 490.577,Z 479.35,A -85,B 0,C 180,E1 -6495.369,E2 -6495.369} C_VEL
LIN {X 0,Y 491.213,Z 466.906,A -85,B 0,C 180,E1 -6496.544,E2 -6496.544} C_VEL
LIN {X 0,Y 491.819,Z 453.636,A -85,B 0,C 180,E1 -6497.57,E2 -6497.57} C_VEL
LIN {X 0,Y 492.348,Z 440.764,A -85,B 0,C 180,E1 -6498.382,E2 -6498.382} C_VEL
LIN {X 0,Y 492.807,Z 426.671,A -85,B 0,C 180,E1 -6499.091,E2 -6499.091} C_VEL
LIN {X 0,Y 488.767,Z 413.231,A -85,B 0,C 180,E1 -6499.804,E2 -6499.804} C_VEL
LIN {X 0,Y 488.711,Z 413.233,A -85,B 0,C 180,E1 -6503.02,E2 -6503.02} C_VEL
LIN {X 0,Y 488.729,Z 413.235,A -85,B 0,C 180,E1 -6505.557,E2 -6505.557} C_VEL
LIN {X 0,Y 488.747,Z 413.232,A -85,B 0,C 180,E1 -6508.329,E2 -6508.329} C_VEL
LIN {X 0,Y 488.696,Z 413.235,A -85,B 0,C 180,E1 -6511.179,E2 -6511.179} C_VEL
LIN {X 0,Y 488.732,Z 413.233,A -85,B 0,C 180,E1 -6514.113,E2 -6514.113} C_VEL
LIN {X 0,Y 488.681,Z 413.238,A -85,B 0,C 180,E1 -6517.159,E2 -6517.159} C_VEL
LIN {X 0,Y 488.719,Z 413.233,A -85,B 0,C 180,E1 -6520.345,E2 -6520.345} C_VEL
LIN {X 0,Y 488.747,Z 413.233,A -85,B 0,C 180,E1 -6523.648,E2 -6523.648} C_VEL
LIN {X 0,Y 488.764,Z 413.255,A -85,B 0,C 180,E1 -6524.168,E2 -6524.168} C_VEL
LIN {X 0,Y 488.933,Z 416.137,A -85,B 0,C 180,E1 -6525.224,E2 -6525.224} C_VEL
LIN {X 0,Y 488.593,Z 427.846,A -85,B 0,C 180,E1 -6529.12,E2 -6529.12} C_VEL
LIN {X 0,Y 488.816,Z 437.833,A -85,B 0,C 180,E1 -6532.257,E2 -6532.257} C_VEL
LIN {X 0,Y 488.983,Z 446.84,A -85,B 0,C 180,E1 -6535.009,E2 -6535.009} C_VEL
LIN {X 0,Y 489.032,Z 456.705,A -85,B 0,C 180,E1 -6537.984,E2 -6537.984} C_VEL
LIN {X 0,Y 489.107,Z 467.512,A -85,B 0,C 180,E1 -6541.224,E2 -6541.224} C_VEL
LIN {X 0,Y 488.908,Z 478.264,A -85,B 0,C 180,E1 -6544.453,E2 -6544.453} C_VEL
LIN {X 0,Y 488.79,Z 487.16,A -85,B 0,C 180,E1 -6547.156,E2 -6547.156} C_VEL
LIN {X 0,Y 488.665,Z 495.726,A -85,B 0,C 180,E1 -6549.808,E2 -6549.808} C_VEL
LIN {X 0,Y 488.496,Z 502.523,A -85,B 0,C 180,E1 -6552.197,E2 -6552.197} C_VEL
LIN {X 0,Y 491.71,Z 517.77,A -85,B 0,C 180,E1 -6552.65,E2 -6552.65} C_VEL
LIN {X 0,Y 492.238,Z 521.762,A -85,B 0,C 180,E1 -6552.786,E2 -6552.786} C_VEL
LIN {X 0,Y 491.896,Z 534.924,A -85,B 0,C 180,E1 -6553.269,E2 -6553.269} C_VEL
LIN {X 0,Y 491.399,Z 548.034,A -85,B 0,C 180,E1 -6553.913,E2 -6553.913} C_VEL
LIN {X 0,Y 490.868,Z 561.231,A -85,B 0,C 180,E1 -6554.747,E2 -6554.747} C_VEL
LIN {X 0,Y 490.251,Z 573.148,A -85,B 0,C 180,E1 -6555.683,E2 -6555.683} C_VEL
LIN {X 0,Y 489.722,Z 584.015,A -85,B 0,C 180,E1 -6556.726,E2 -6556.726} C_VEL
LIN {X 0,Y 489.274,Z 594.068,A -85,B 0,C 180,E1 -6557.891,E2 -6557.891} C_VEL
LIN {X 0,Y 488.839,Z 603.576,A -85,B 0,C 180,E1 -6559.228,E2 -6559.228} C_VEL
LIN {X 0,Y 488.463,Z 612.023,A -85,B 0,C 180,E1 -6560.685,E2 -6560.685} C_VEL
LIN {X 0,Y 488.192,Z 618.847,A -85,B 0,C 180,E1 -6562.139,E2 -6562.139} C_VEL
LIN {X 0,Y 488.038,Z 624.897,A -85,B 0,C 180,E1 -6563.78,E2 -6563.78} C_VEL
LIN {X 0,Y 487.962,Z 628.441,A -85,B 0,C 180,E1 -6565.043,E2 -6565.043} C_VEL
LIN {X 0,Y 487.956,Z 631.826,A -85,B 0,C 180,E1 -6566.697,E2 -6566.697} C_VEL
LIN {X 0,Y 487.885,Z 633.83,A -85,B 0,C 180,E1 -6568.349,E2 -6568.349} C_VEL
LIN {X 0,Y 487.817,Z 634.5,A -85,B 0,C 180,E1 -6570,E2 -6570} C_VEL
LIN {X 0,Y 487.885,Z 633.827,A -85,B 0,C 180,E1 -6571.651,E2 -6571.651} C_VEL
LIN {X 0,Y 487.956,Z 631.826,A -85,B 0,C 180,E1 -6573.303,E2 -6573.303} C_VEL
LIN {X 0,Y 487.962,Z 628.446,A -85,B 0,C 180,E1 -6574.958,E2 -6574.958} C_VEL
LIN {X 0,Y 488.047,Z 624.051,A -85,B 0,C 180,E1 -6576.477,E2 -6576.477} C_VEL
LIN {X 0,Y 488.193,Z 618.861,A -85,B 0,C 180,E1 -6577.861,E2 -6577.861} C_VEL
LIN {X 0,Y 488.477,Z 612.056,A -85,B 0,C 180,E1 -6579.315,E2 -6579.315} C_VEL
LIN {X 0,Y 488.837,Z 603.57,A -85,B 0,C 180,E1 -6580.772,E2 -6580.772} C_VEL
LIN {X 0,Y 489.253,Z 594.237,A -85,B 0,C 180,E1 -6582.083,E2 -6582.083} C_VEL
LIN {X 0,Y 489.731,Z 583.991,A -85,B 0,C 180,E1 -6583.274,E2 -6583.274} C_VEL
LIN {X 0,Y 490.251,Z 573.157,A -85,B 0,C 180,E1 -6584.317,E2 -6584.317} C_VEL
LIN {X 0,Y 490.867,Z 561.271,A -85,B 0,C 180,E1 -6585.253,E2 -6585.253} C_VEL
LIN {X 0,Y 491.411,Z 548.036,A -85,B 0,C 180,E1 -6586.087,E2 -6586.087} C_VEL
LIN {X 0,Y 491.903,Z 534.341,A -85,B 0,C 180,E1 -6586.755,E2 -6586.755} C_VEL
LIN {X 0,Y 492.168,Z 520.053,A -85,B 0,C 180,E1 -6587.27,E2 -6587.27} C_VEL
LIN {X 0,Y 489.106,Z 505.352,A -85,B 0,C 180,E1 -6587.73,E2 -6587.73} C_VEL
LIN {X 0,Y 488.508,Z 502.42,A -85,B 0,C 180,E1 -6587.829,E2 -6587.829} C_VEL
LIN {X 0,Y 488.674,Z 493.906,A -85,B 0,C 180,E1 -6590.802,E2 -6590.802} C_VEL
LIN {X 0,Y 488.865,Z 485.166,A -85,B 0,C 180,E1 -6593.737,E2 -6593.737} C_VEL
LIN {X 0,Y 489.02,Z 477.15,A -85,B 0,C 180,E1 -6596.457,E2 -6596.457} C_VEL
LIN {X 0,Y 489.279,Z 469.264,A -85,B 0,C 180,E1 -6599.234,E2 -6599.234} C_VEL
LIN {X 0,Y 489.457,Z 459.984,A -85,B 0,C 180,E1 -6602.578,E2 -6602.578} C_VEL
LIN {X 0,Y 489.657,Z 452.009,A -85,B 0,C 180,E1 -6605.541,E2 -6605.541} C_VEL
LIN {X 0,Y 489.802,Z 444.051,A -85,B 0,C 180,E1 -6608.621,E2 -6608.621} C_VEL
LIN {X 0,Y 489.996,Z 437.39,A -85,B 0,C 180,E1 -6611.283,E2 -6611.283} C_VEL
LIN {X 0,Y 490.317,Z 429.32,A -85,B 0,C 180,E1 -6614.616,E2 -6614.616} C_VEL
LIN {X 0,Y 490.414,Z 423.879,A -85,B 0,C 180,E1 -6616.959,E2 -6616.959} C_VEL
LIN {X 0,Y 489.632,Z 418.296,A -85,B 0,C 180,E1 -6619.53,E2 -6619.53} C_VEL
LIN {X 0,Y 488.733,Z 413.234,A -85,B 0,C 180,E1 -6622.077,E2 -6622.077} C_VEL
LIN {X 0,Y 488.729,Z 413.233,A -85,B 0,C 180,E1 -6625.052,E2 -6625.052} C_VEL
LIN {X 0,Y 488.705,Z 413.237,A -85,B 0,C 180,E1 -6628.046,E2 -6628.046} C_VEL
LIN {X 0,Y 488.725,Z 413.233,A -85,B 0,C 180,E1 -6630.73,E2 -6630.73} C_VEL
LIN {X 0,Y 488.759,Z 413.221,A -85,B 0,C 180,E1 -6633.528,E2 -6633.528} C_VEL
LIN {X 0,Y 488.696,Z 413.237,A -85,B 0,C 180,E1 -6636.255,E2 -6636.255} C_VEL
LIN {X 0,Y 488.748,Z 413.223,A -85,B 0,C 180,E1 -6639.176,E2 -6639.176} C_VEL
LIN {X 0,Y 488.761,Z 413.228,A -85,B 0,C 180,E1 -6641.628,E2 -6641.628} C_VEL
LIN {X 0,Y 488.764,Z 413.222,A -85,B 0,C 180,E1 -6645,E2 -6645} C_VEL
LIN {X 0,Y 488.808,Z 413.222,A -85,B 0,C 180,E1 -6648.388,E2 -6648.388} C_VEL
LIN {X 0,Y 488.788,Z 413.218,A -85,B 0,C 180,E1 -6651.733,E2 -6651.733} C_VEL
LIN {X 0,Y 488.858,Z 413.217,A -85,B 0,C 180,E1 -6654.224,E2 -6654.224} C_VEL
LIN {X 0,Y 488.963,Z 413.197,A -85,B 0,C 180,E1 -6657.529,E2 -6657.529} C_VEL
LIN {X 0,Y 488.957,Z 413.202,A -85,B 0,C 180,E1 -6660.824,E2 -6660.824} C_VEL
LIN {X 0,Y 488.962,Z 413.198,A -85,B 0,C 180,E1 -6662.471,E2 -6662.471} C_VEL
LIN {X 0,Y 488.857,Z 413.217,A -85,B 0,C 180,E1 -6665.776,E2 -6665.776} C_VEL
LIN {X 0,Y 488.82,Z 413.213,A -85,B 0,C 180,E1 -6668.266,E2 -6668.266} C_VEL
LIN {X 0,Y 488.808,Z 413.223,A -85,B 0,C 180,E1 -6671.612,E2 -6671.612} C_VEL
LIN {X 0,Y 488.764,Z 413.227,A -85,B 0,C 180,E1 -6675,E2 -6675} C_VEL
LIN {X 0,Y 488.757,Z 413.224,A -85,B 0,C 180,E1 -6678.442,E2 -6678.442} C_VEL
LIN {X 0,Y 488.709,Z 413.238,A -85,B 0,C 180,E1 -6681.071,E2 -6681.071} C_VEL
LIN {X 0,Y 488.682,Z 413.235,A -85,B 0,C 180,E1 -6683.746,E2 -6683.746} C_VEL
LIN {X 0,Y 488.794,Z 413.223,A -85,B 0,C 180,E1 -6686.944,E2 -6686.944} C_VEL
LIN {X 0,Y 488.712,Z 413.235,A -85,B 0,C 180,E1 -6690.363,E2 -6690.363} C_VEL
LIN {X 0,Y 488.736,Z 413.232,A -85,B 0,C 180,E1 -6693.484,E2 -6693.484} C_VEL
LIN {X 0,Y 488.684,Z 413.24,A -85,B 0,C 180,E1 -6696.355,E2 -6696.355} C_VEL
LIN {X 0,Y 488.703,Z 413.237,A -85,B 0,C 180,E1 -6699.254,E2 -6699.254} C_VEL
LIN {X 0,Y 488.725,Z 413.233,A -85,B 0,C 180,E1 -6701.602,E2 -6701.602} C_VEL
LIN {X 0,Y 488.714,Z 413.235,A -85,B 0,C 180,E1 -6704.801,E2 -6704.801} C_VEL
LIN {X 0,Y 488.694,Z 413.24,A -85,B 0,C 180,E1 -6707.475,E2 -6707.475} C_VEL
LIN {X 0,Y 488.778,Z 413.364,A -85,B 0,C 180,E1 -6709.485,E2 -6709.485} C_VEL
LIN {X 0,Y 489.889,Z 419.839,A -85,B 0,C 180,E1 -6711.387,E2 -6711.387} C_VEL
LIN {X 0,Y 489.973,Z 425.259,A -85,B 0,C 180,E1 -6712.956,E2 -6712.956} C_VEL
LIN {X 0,Y 489.646,Z 436.842,A -85,B 0,C 180,E1 -6716.355,E2 -6716.355} C_VEL
LIN {X 0,Y 489.545,Z 445.302,A -85,B 0,C 180,E1 -6718.881,E2 -6718.881} C_VEL
LIN {X 0,Y 489.375,Z 456.104,A -85,B 0,C 180,E1 -6722.106,E2 -6722.106} C_VEL
LIN {X 0,Y 488.651,Z 458.349,A -85,B 0,C 180,E1 -6722.74,E2 -6722.74} C_VEL
LIN {X 0,Y 482.752,Z 466.151,A -85,B 0,C 180,E1 -6724.782,E2 -6724.782} C_VEL
LIN {X 0,Y 482.025,Z 468.434,A -85,B 0,C 180,E1 -6725.427,E2 -6725.427} C_VEL
LIN {X 0,Y 481.869,Z 477.854,A -85,B 0,C 180,E1 -6728.166,E2 -6728.166} C_VEL
LIN {X 0,Y 481.668,Z 488.876,A -85,B 0,C 180,E1 -6731.276,E2 -6731.276} C_VEL
LIN {X 0,Y 481.64,Z 491.377,A -85,B 0,C 180,E1 -6731.968,E2 -6731.968} C_VEL
LIN {X 0,Y 484.961,Z 507.326,A -85,B 0,C 180,E1 -6732.435,E2 -6732.435} C_VEL
LIN {X 0,Y 485.491,Z 511.317,A -85,B 0,C 180,E1 -6732.574,E2 -6732.574} C_VEL
LIN {X 0,Y 485.096,Z 524.157,A -85,B 0,C 180,E1 -6733.038,E2 -6733.038} C_VEL
LIN {X 0,Y 484.664,Z 537.399,A -85,B 0,C 180,E1 -6733.683,E2 -6733.683} C_VEL
LIN {X 0,Y 484.106,Z 549.31,A -85,B 0,C 180,E1 -6734.421,E2 -6734.421} C_VEL
LIN {X 0,Y 483.509,Z 560.39,A -85,B 0,C 180,E1 -6735.264,E2 -6735.264} C_VEL
LIN {X 0,Y 482.94,Z 571.788,A -85,B 0,C 180,E1 -6736.321,E2 -6736.321} C_VEL
LIN {X 0,Y 482.414,Z 581.804,A -85,B 0,C 180,E1 -6737.444,E2 -6737.444} C_VEL
LIN {X 0,Y 482.05,Z 590.748,A -85,B 0,C 180,E1 -6738.649,E2 -6738.649} C_VEL
LIN {X 0,Y 481.588,Z 598.624,A -85,B 0,C 180,E1 -6739.914,E2 -6739.914} C_VEL
LIN {X 0,Y 481.319,Z 605.179,A -85,B 0,C 180,E1 -6741.181,E2 -6741.181} C_VEL
LIN {X 0,Y 481.059,Z 610.622,A -85,B 0,C 180,E1 -6742.445,E2 -6742.445} C_VEL
LIN {X 0,Y 480.986,Z 616.321,A -85,B 0,C 180,E1 -6744.129,E2 -6744.129} C_VEL
LIN {X 0,Y 480.821,Z 620.47,A -85,B 0,C 180,E1 -6745.809,E2 -6745.809} C_VEL
LIN {X 0,Y 480.881,Z 622,A -85,B 0,C 180,E1 -6746.649,E2 -6746.649} C_VEL
LIN {X 0,Y 480.788,Z 624.036,A -85,B 0,C 180,E1 -6748.325,E2 -6748.325} C_VEL
LIN {X 0,Y 480.742,Z 624.741,A -85,B 0,C 180,E1 -6750,E2 -6750} C_VEL
LIN {X 0,Y 480.787,Z 624.117,A -85,B 0,C 180,E1 -6751.675,E2 -6751.675} C_VEL
LIN {X 0,Y 480.88,Z 622.15,A -85,B 0,C 180,E1 -6753.351,E2 -6753.351} C_VEL
LIN {X 0,Y 480.899,Z 618.802,A -85,B 0,C 180,E1 -6755.03,E2 -6755.03} C_VEL
LIN {X 0,Y 481.01,Z 613.975,A -85,B 0,C 180,E1 -6756.713,E2 -6756.713} C_VEL
LIN {X 0,Y 481.224,Z 607.518,A -85,B 0,C 180,E1 -6758.398,E2 -6758.398} C_VEL
LIN {X 0,Y 481.534,Z 600.322,A -85,B 0,C 180,E1 -6759.875,E2 -6759.875} C_VEL
LIN {X 0,Y 482.004,Z 591.365,A -85,B 0,C 180,E1 -6761.352,E2 -6761.352} C_VEL
LIN {X 0,Y 482.438,Z 581.993,A -85,B 0,C 180,E1 -6762.622,E2 -6762.622} C_VEL
LIN {X 0,Y 482.982,Z 571.621,A -85,B 0,C 180,E1 -6763.785,E2 -6763.785} C_VEL
LIN {X 0,Y 483.542,Z 560.182,A -85,B 0,C 180,E1 -6764.843,E2 -6764.843} C_VEL
LIN {X 0,Y 484.192,Z 547.519,A -85,B 0,C 180,E1 -6765.793,E2 -6765.793} C_VEL
LIN {X 0,Y 484.756,Z 534.202,A -85,B 0,C 180,E1 -6766.585,E2 -6766.585} C_VEL
LIN {X 0,Y 485.207,Z 520.421,A -85,B 0,C 180,E1 -6767.206,E2 -6767.206} C_VEL
LIN {X 0,Y 485.413,Z 509.833,A -85,B 0,C 180,E1 -6767.566,E2 -6767.566} C_VEL
LIN {X 0,Y 482.421,Z 495.181,A -85,B 0,C 180,E1 -6768.027,E2 -6768.027} C_VEL
LIN {X 0,Y 481.631,Z 491.328,A -85,B 0,C 180,E1 -6768.135,E2 -6768.135} C_VEL
LIN {X 0,Y 481.846,Z 479.736,A -85,B 0,C 180,E1 -6771.385,E2 -6771.385} C_VEL
LIN {X 0,Y 482.015,Z 468.814,A -85,B 0,C 180,E1 -6774.554,E2 -6774.554} C_VEL
LIN {X 0,Y 482.327,Z 457.914,A -85,B 0,C 180,E1 -6777.793,E2 -6777.793} C_VEL
LIN {X 0,Y 482.54,Z 446.788,A -85,B 0,C 180,E1 -6781.14,E2 -6781.14} C_VEL
LIN {X 0,Y 482.677,Z 436.617,A -85,B 0,C 180,E1 -6784.207,E2 -6784.207} C_VEL
LIN {X 0,Y 483.071,Z 424.92,A -85,B 0,C 180,E1 -6787.665,E2 -6787.665} C_VEL
LIN {X 0,Y 482.742,Z 420.055,A -85,B 0,C 180,E1 -6789.104,E2 -6789.104} C_VEL
LIN {X 0,Y 481.711,Z 414.111,A -85,B 0,C 180,E1 -6790.923,E2 -6790.923} C_VEL
LIN {X 0,Y 481.662,Z 414.116,A -85,B 0,C 180,E1 -6794.457,E2 -6794.457} C_VEL
LIN {X 0,Y 481.68,Z 414.114,A -85,B 0,C 180,E1 -6796.847,E2 -6796.847} C_VEL
LIN {X 0,Y 481.678,Z 414.114,A -85,B 0,C 180,E1 -6800.06,E2 -6800.06} C_VEL
LIN {X 0,Y 481.631,Z 414.117,A -85,B 0,C 180,E1 -6803.253,E2 -6803.253} C_VEL
LIN {X 0,Y 481.712,Z 414.103,A -85,B 0,C 180,E1 -6806.33,E2 -6806.33} C_VEL
LIN {X 0,Y 481.66,Z 414.108,A -85,B 0,C 180,E1 -6809.416,E2 -6809.416} C_VEL
LIN {X 0,Y 481.703,Z 414.108,A -85,B 0,C 180,E1 -6812.168,E2 -6812.168} C_VEL
LIN {X 0,Y 481.721,Z 414.107,A -85,B 0,C 180,E1 -6814.97,E2 -6814.97} C_VEL
LIN {X 0,Y 481.653,Z 414.115,A -85,B 0,C 180,E1 -6817.705,E2 -6817.705} C_VEL
LIN {X 0,Y 481.686,Z 414.113,A -85,B 0,C 180,E1 -6819.948,E2 -6819.948} C_VEL
LIN {X 0,Y 485.897,Z 427.235,A -85,B 0,C 180,E1 -6820.694,E2 -6820.694} C_VEL
LIN {X 0,Y 486.087,Z 429.854,A -85,B 0,C 180,E1 -6820.831,E2 -6820.831} C_VEL
LIN {X 0,Y 485.581,Z 442.838,A -85,B 0,C 180,E1 -6821.542,E2 -6821.542} C_VEL
LIN {X 0,Y 484.863,Z 456.913,A -85,B 0,C 180,E1 -6822.496,E2 -6822.496} C_VEL
LIN {X 0,Y 484.179,Z 470.077,A -85,B 0,C 180,E1 -6823.596,E2 -6823.596} C_VEL
LIN {X 0,Y 483.607,Z 480.35,A -85,B 0,C 180,E1 -6824.62,E2 -6824.62} C_VEL
LIN {X 0,Y 483.047,Z 491.164,A -85,B 0,C 180,E1 -6825.895,E2 -6825.895} C_VEL
LIN {X 0,Y 482.477,Z 500.306,A -85,B 0,C 180,E1 -6827.165,E2 -6827.165} C_VEL
LIN {X 0,Y 482.108,Z 509.218,A -85,B 0,C 180,E1 -6828.65,E2 -6828.65} C_VEL
LIN {X 0,Y 481.588,Z 517.54,A -85,B 0,C 180,E1 -6830.339,E2 -6830.339} C_VEL
LIN {X 0,Y 481.364,Z 524.181,A -85,B 0,C 180,E1 -6832.027,E2 -6832.027} C_VEL
LIN {X 0,Y 481.15,Z 529.201,A -85,B 0,C 180,E1 -6833.641,E2 -6833.641} C_VEL
LIN {X 0,Y 481.073,Z 532.37,A -85,B 0,C 180,E1 -6834.971,E2 -6834.971} C_VEL
LIN {X 0,Y 481.009,Z 535.324,A -85,B 0,C 180,E1 -6836.649,E2 -6836.649} C_VEL
LIN {X 0,Y 480.882,Z 537.123,A -85,B 0,C 180,E1 -6838.325,E2 -6838.325} C_VEL
LIN {X 0,Y 480.838,Z 537.787,A -85,B 0,C 180,E1 -6840,E2 -6840} C_VEL
